LIN {X 0,Y 419.187,Z 570.974,A -85,B 0,C 180,E1 -10319.804,E2 -10319.804} C_VEL
LIN {X 0,Y 418.475,Z 578.407,A -85,B 0,C 180,E1 -10321.405,E2 -10321.405} C_VEL
LIN {X 0,Y 417.933,Z 584.546,A -85,B 0,C 180,E1 -10323.03,E2 -10323.03} C_VEL
LIN {X 0,Y 417.578,Z 589.288,A -85,B 0,C 180,E1 -10324.586,E2 -10324.586} C_VEL
LIN {X 0,Y 417.334,Z 593.011,A -85,B 0,C 180,E1 -10326.162,E2 -10326.162} C_VEL
LIN {X 0,Y 417.085,Z 596.065,A -85,B 0,C 180,E1 -10327.935,E2 -10327.935} C_VEL
LIN {X 0,Y 416.98,Z 597.612,A -85,B 0,C 180,E1 -10329.272,E2 -10329.272} C_VEL
LIN {X 0,Y 416.926,Z 598.729,A -85,B 0,C 180,E1 -10331.321,E2 -10331.321} C_VEL
LIN {X 0,Y 416.921,Z 598.396,A -85,B 0,C 180,E1 -10333.348,E2 -10333.348} C_VEL
LIN {X 0,Y 416.982,Z 596.643,A -85,B 0,C 180,E1 -10335.357,E2 -10335.357} C_VEL
LIN {X 0,Y 417.194,Z 593.458,A -85,B 0,C 180,E1 -10337.351,E2 -10337.351} C_VEL
LIN {X 0,Y 417.313,Z 591.479,A -85,B 0,C 180,E1 -10338.264,E2 -10338.264} C_VEL
LIN {X 0,Y 416.787,Z 589.683,A -85,B 0,C 180,E1 -10339.033,E2 -10339.033} C_VEL
LIN {X 0,Y 414.202,Z 586.34,A -85,B 0,C 180,E1 -10340.269,E2 -10340.269} C_VEL
LIN {X 0,Y 411.626,Z 582.374,A -85,B 0,C 180,E1 -10341.484,E2 -10341.484} C_VEL
LIN {X 0,Y 411.128,Z 579.597,A -85,B 0,C 180,E1 -10342.211,E2 -10342.211} C_VEL
LIN {X 0,Y 411.667,Z 572.14,A -85,B 0,C 180,E1 -10343.876,E2 -10343.876} C_VEL
LIN {X 0,Y 412.417,Z 564.039,A -85,B 0,C 180,E1 -10345.358,E2 -10345.358} C_VEL
LIN {X 0,Y 413.292,Z 554.296,A -85,B 0,C 180,E1 -10346.833,E2 -10346.833} C_VEL
LIN {X 0,Y 414.16,Z 543.524,A -85,B 0,C 180,E1 -10348.178,E2 -10348.178} C_VEL
LIN {X 0,Y 415.25,Z 531.337,A -85,B 0,C 180,E1 -10349.414,E2 -10349.414} C_VEL
LIN {X 0,Y 416.092,Z 519.779,A -85,B 0,C 180,E1 -10350.364,E2 -10350.364} C_VEL
LIN {X 0,Y 416.915,Z 506.934,A -85,B 0,C 180,E1 -10351.208,E2 -10351.208} C_VEL
LIN {X 0,Y 417.627,Z 493.022,A -85,B 0,C 180,E1 -10351.899,E2 -10351.899} C_VEL
LIN {X 0,Y 418.129,Z 479.426,A -85,B 0,C 180,E1 -10352.379,E2 -10352.379} C_VEL
LIN {X 0,Y 418.499,Z 462.629,A -85,B 0,C 180,E1 -10352.738,E2 -10352.738} C_VEL
LIN {X 0,Y 419.9,Z 361.135,A -85,B 0,C 180,E1 -10354.504,E2 -10354.504} C_VEL
LIN {X 0,Y 416.679,Z 347.393,A -85,B 0,C 180,E1 -10354.918,E2 -10354.918} C_VEL
LIN {X 0,Y 413.389,Z 338.049,A -85,B 0,C 180,E1 -10355.274,E2 -10355.274} C_VEL
LIN {X 0,Y 411.415,Z 327.865,A -85,B 0,C 180,E1 -10357.64,E2 -10357.64} C_VEL
LIN {X 0,Y 411.281,Z 327.882,A -85,B 0,C 180,E1 -10360.835,E2 -10360.835} C_VEL
LIN {X 0,Y 411.251,Z 327.88,A -85,B 0,C 180,E1 -10363.843,E2 -10363.843} C_VEL
LIN {X 0,Y 411.256,Z 327.881,A -85,B 0,C 180,E1 -10366.89,E2 -10366.89} C_VEL
LIN {X 0,Y 411.23,Z 327.882,A -85,B 0,C 180,E1 -10369.988,E2 -10369.988} C_VEL
LIN {X 0,Y 411.186,Z 327.894,A -85,B 0,C 180,E1 -10373.149,E2 -10373.149} C_VEL
LIN {X 0,Y 411.17,Z 327.89,A -85,B 0,C 180,E1 -10376.386,E2 -10376.386} C_VEL
LIN {X 0,Y 411.193,Z 327.887,A -85,B 0,C 180,E1 -10379.714,E2 -10379.714} C_VEL
LIN {X 0,Y 411.201,Z 327.89,A -85,B 0,C 180,E1 -10383.157,E2 -10383.157} C_VEL
LIN {X 0,Y 411.187,Z 327.89,A -85,B 0,C 180,E1 -10386.552,E2 -10386.552} C_VEL
LIN {X 0,Y 411.167,Z 327.889,A -85,B 0,C 180,E1 -10389.721,E2 -10389.721} C_VEL
LIN {X 0,Y 411.16,Z 327.893,A -85,B 0,C 180,E1 -10393.136,E2 -10393.136} C_VEL
LIN {X 0,Y 411.162,Z 327.89,A -85,B 0,C 180,E1 -10395.883,E2 -10395.883} C_VEL
LIN {X 0,Y 411.156,Z 327.891,A -85,B 0,C 180,E1 -10399.493,E2 -10399.493} C_VEL
LIN {X 0,Y 411.177,Z 327.889,A -85,B 0,C 180,E1 -10402.025,E2 -10402.025} C_VEL
LIN {X 0,Y 411.201,Z 327.886,A -85,B 0,C 180,E1 -10405.124,E2 -10405.124} C_VEL
LIN {X 0,Y 411.164,Z 327.891,A -85,B 0,C 180,E1 -10408.003,E2 -10408.003} C_VEL
LIN {X 0,Y 411.172,Z 327.889,A -85,B 0,C 180,E1 -10411.407,E2 -10411.407} C_VEL
LIN {X 0,Y 411.189,Z 327.888,A -85,B 0,C 180,E1 -10414.942,E2 -10414.942} C_VEL
LIN {X 0,Y 411.202,Z 327.887,A -85,B 0,C 180,E1 -10417.914,E2 -10417.914} C_VEL
LIN {X 0,Y 411.216,Z 327.884,A -85,B 0,C 180,E1 -10421.052,E2 -10421.052} C_VEL
LIN {X 0,Y 411.213,Z 327.889,A -85,B 0,C 180,E1 -10424.13,E2 -10424.13} C_VEL
LIN {X 0,Y 411.306,Z 327.872,A -85,B 0,C 180,E1 -10427.166,E2 -10427.166} C_VEL
LIN {X 0,Y 411.293,Z 327.881,A -85,B 0,C 180,E1 -10430.162,E2 -10430.162} C_VEL
LIN {X 0,Y 411.397,Z 327.861,A -85,B 0,C 180,E1 -10433.132,E2 -10433.132} C_VEL
LIN {X 0,Y 411.303,Z 327.872,A -85,B 0,C 180,E1 -10435.099,E2 -10435.099} C_VEL
LIN {X 0,Y 411.512,Z 327.853,A -85,B 0,C 180,E1 -10438.043,E2 -10438.043} C_VEL
LIN {X 0,Y 411.636,Z 327.838,A -85,B 0,C 180,E1 -10440,E2 -10440} C_VEL
LIN {X 0,Y 411.448,Z 327.854,A -85,B 0,C 180,E1 -10442.938,E2 -10442.938} C_VEL
LIN {X 0,Y 411.462,Z 327.86,A -85,B 0,C 180,E1 -10445.883,E2 -10445.883} C_VEL
LIN {X 0,Y 411.337,Z 327.868,A -85,B 0,C 180,E1 -10448.846,E2 -10448.846} C_VEL
LIN {X 0,Y 411.287,Z 327.881,A -85,B 0,C 180,E1 -10451.833,E2 -10451.833} C_VEL
LIN {X 0,Y 411.263,Z 327.877,A -85,B 0,C 180,E1 -10454.853,E2 -10454.853} C_VEL
LIN {X 0,Y 411.256,Z 327.883,A -85,B 0,C 180,E1 -10457.915,E2 -10457.915} C_VEL
LIN {X 0,Y 411.201,Z 327.886,A -85,B 0,C 180,E1 -10461.034,E2 -10461.034} C_VEL
LIN {X 0,Y 411.23,Z 327.882,A -85,B 0,C 180,E1 -10464.216,E2 -10464.216} C_VEL
LIN {X 0,Y 411.263,Z 327.884,A -85,B 0,C 180,E1 -10467.478,E2 -10467.478} C_VEL
LIN {X 0,Y 411.193,Z 327.887,A -85,B 0,C 180,E1 -10470.848,E2 -10470.848} C_VEL
LIN {X 0,Y 411.209,Z 327.884,A -85,B 0,C 180,E1 -10474.333,E2 -10474.333} C_VEL
LIN {X 0,Y 411.199,Z 327.886,A -85,B 0,C 180,E1 -10477.974,E2 -10477.974} C_VEL
LIN {X 0,Y 411.186,Z 327.887,A -85,B 0,C 180,E1 -10480.504,E2 -10480.504} C_VEL
LIN {X 0,Y 411.181,Z 327.893,A -85,B 0,C 180,E1 -10483.133,E2 -10483.133} C_VEL
LIN {X 0,Y 411.173,Z 327.889,A -85,B 0,C 180,E1 -10485.881,E2 -10485.881} C_VEL
LIN {X 0,Y 411.167,Z 327.892,A -85,B 0,C 180,E1 -10488.771,E2 -10488.771} C_VEL
LIN {X 0,Y 411.209,Z 327.885,A -85,B 0,C 180,E1 -10491.831,E2 -10491.831} C_VEL
LIN {X 0,Y 411.215,Z 327.89,A -85,B 0,C 180,E1 -10495.121,E2 -10495.121} C_VEL
LIN {X 0,Y 411.17,Z 327.895,A -85,B 0,C 180,E1 -10498.002,E2 -10498.002} C_VEL
LIN {X 0,Y 411.253,Z 327.986,A -85,B 0,C 180,E1 -10499.548,E2 -10499.548} C_VEL
LIN {X 0,Y 415.143,Z 345.403,A -85,B 0,C 180,E1 -10503.042,E2 -10503.042} C_VEL
LIN {X 0,Y 415.639,Z 350.042,A -85,B 0,C 180,E1 -10503.919,E2 -10503.919} C_VEL
LIN {X 0,Y 414.463,Z 366.202,A -85,B 0,C 180,E1 -10506.786,E2 -10506.786} C_VEL
LIN {X 0,Y 419.646,Z 398,A -85,B 0,C 180,E1 -10507.644,E2 -10507.644} C_VEL
LIN {X 0,Y 417.994,Z 504.817,A -85,B 0,C 180,E1 -10509.516,E2 -10509.516} C_VEL
LIN {X 0,Y 417.425,Z 519.405,A -85,B 0,C 180,E1 -10509.969,E2 -10509.969} C_VEL
LIN {X 0,Y 416.661,Z 532.568,A -85,B 0,C 180,E1 -10510.558,E2 -10510.558} C_VEL
LIN {X 0,Y 415.788,Z 546.414,A -85,B 0,C 180,E1 -10511.394,E2 -10511.394} C_VEL
LIN {X 0,Y 414.754,Z 559.052,A -85,B 0,C 180,E1 -10512.368,E2 -10512.368} C_VEL
LIN {X 0,Y 413.786,Z 570.591,A -85,B 0,C 180,E1 -10513.471,E2 -10513.471} C_VEL
LIN {X 0,Y 412.832,Z 581.181,A -85,B 0,C 180,E1 -10514.699,E2 -10514.699} C_VEL
LIN {X 0,Y 412.026,Z 591.716,A -85,B 0,C 180,E1 -10516.183,E2 -10516.183} C_VEL
LIN {X 0,Y 411.345,Z 600.394,A -85,B 0,C 180,E1 -10517.668,E2 -10517.668} C_VEL
LIN {X 0,Y 410.689,Z 608.675,A -85,B 0,C 180,E1 -10519.399,E2 -10519.399} C_VEL
LIN {X 0,Y 410.326,Z 615.336,A -85,B 0,C 180,E1 -10521.132,E2 -10521.132} C_VEL
LIN {X 0,Y 410.062,Z 621.237,A -85,B 0,C 180,E1 -10523.109,E2 -10523.109} C_VEL
LIN {X 0,Y 409.983,Z 625.54,A -85,B 0,C 180,E1 -10525.082,E2 -10525.082} C_VEL
LIN {X 0,Y 409.955,Z 628.378,A -85,B 0,C 180,E1 -10527.051,E2 -10527.051} C_VEL
LIN {X 0,Y 409.954,Z 629.831,A -85,B 0,C 180,E1 -10529.017,E2 -10529.017} C_VEL
LIN {X 0,Y 409.954,Z 629.934,A -85,B 0,C 180,E1 -10530.981,E2 -10530.981} C_VEL
LIN {X 0,Y 409.994,Z 629.483,A -85,B 0,C 180,E1 -10531.964,E2 -10531.964} C_VEL
LIN {X 0,Y 409.922,Z 627.565,A -85,B 0,C 180,E1 -10533.931,E2 -10533.931} C_VEL
LIN {X 0,Y 410.015,Z 624.244,A -85,B 0,C 180,E1 -10535.902,E2 -10535.902} C_VEL
LIN {X 0,Y 410.154,Z 620.769,A -85,B 0,C 180,E1 -10537.383,E2 -10537.383} C_VEL
LIN {X 0,Y 410.472,Z 614.788,A -85,B 0,C 180,E1 -10539.36,E2 -10539.36} C_VEL
LIN {X 0,Y 410.951,Z 608.074,A -85,B 0,C 180,E1 -10541.092,E2 -10541.092} C_VEL
LIN {X 0,Y 411.639,Z 599.741,A -85,B 0,C 180,E1 -10542.823,E2 -10542.823} C_VEL
LIN {X 0,Y 412.437,Z 591.079,A -85,B 0,C 180,E1 -10544.304,E2 -10544.304} C_VEL
LIN {X 0,Y 413.43,Z 580.609,A -85,B 0,C 180,E1 -10545.782,E2 -10545.782} C_VEL
LIN {X 0,Y 414.659,Z 568.924,A -85,B 0,C 180,E1 -10547.126,E2 -10547.126} C_VEL
LIN {X 0,Y 415.755,Z 557.26,A -85,B 0,C 180,E1 -10548.223,E2 -10548.223} C_VEL
LIN {X 0,Y 416.929,Z 544.33,A -85,B 0,C 180,E1 -10549.197,E2 -10549.197} C_VEL
LIN {X 0,Y 417.819,Z 531.185,A -85,B 0,C 180,E1 -10549.978,E2 -10549.978} C_VEL
LIN {X 0,Y 418.734,Z 517.564,A -85,B 0,C 180,E1 -10550.573,E2 -10550.573} C_VEL
LIN {X 0,Y 419.385,Z 503.626,A -85,B 0,C 180,E1 -10550.989,E2 -10550.989} C_VEL
LIN {X 0,Y 421.169,Z 397.55,A -85,B 0,C 180,E1 -10552.879,E2 -10552.879} C_VEL
LIN {X 0,Y 416.853,Z 373.266,A -85,B 0,C 180,E1 -10553.621,E2 -10553.621} C_VEL
LIN {X 0,Y 415.311,Z 365.541,A -85,B 0,C 180,E1 -10553.906,E2 -10553.906} C_VEL
LIN {X 0,Y 416.42,Z 351.139,A -85,B 0,C 180,E1 -10556.556,E2 -10556.556} C_VEL
LIN {X 0,Y 414.822,Z 342.635,A -85,B 0,C 180,E1 -10558.318,E2 -10558.318} C_VEL
LIN {X 0,Y 412.132,Z 331.458,A -85,B 0,C 180,E1 -10560.768,E2 -10560.768} C_VEL
LIN {X 0,Y 411.159,Z 327.894,A -85,B 0,C 180,E1 -10561.594,E2 -10561.594} C_VEL
LIN {X 0,Y 411.209,Z 327.892,A -85,B 0,C 180,E1 -10564.878,E2 -10564.878} C_VEL
LIN {X 0,Y 411.211,Z 327.886,A -85,B 0,C 180,E1 -10568.169,E2 -10568.169} C_VEL
LIN {X 0,Y 411.196,Z 327.885,A -85,B 0,C 180,E1 -10571.233,E2 -10571.233} C_VEL
LIN {X 0,Y 411.173,Z 327.893,A -85,B 0,C 180,E1 -10574.489,E2 -10574.489} C_VEL
LIN {X 0,Y 411.179,Z 327.893,A -85,B 0,C 180,E1 -10578.194,E2 -10578.194} C_VEL
LIN {X 0,Y 411.213,Z 327.876,A -85,B 0,C 180,E1 -10580.775,E2 -10580.775} C_VEL
LIN {X 0,Y 411.194,Z 327.889,A -85,B 0,C 180,E1 -10584.47,E2 -10584.47} C_VEL
LIN {X 0,Y 411.162,Z 327.891,A -85,B 0,C 180,E1 -10588.002,E2 -10588.002} C_VEL
LIN {X 0,Y 411.217,Z 327.884,A -85,B 0,C 180,E1 -10591.41,E2 -10591.41} C_VEL
LIN {X 0,Y 411.229,Z 327.885,A -85,B 0,C 180,E1 -10594.706,E2 -10594.706} C_VEL
LIN {X 0,Y 411.197,Z 327.885,A -85,B 0,C 180,E1 -10597.913,E2 -10597.913} C_VEL
LIN {X 0,Y 411.217,Z 327.878,A -85,B 0,C 180,E1 -10601.051,E2 -10601.051} C_VEL
LIN {X 0,Y 411.255,Z 327.879,A -85,B 0,C 180,E1 -10604.131,E2 -10604.131} C_VEL
LIN {X 0,Y 411.295,Z 327.875,A -85,B 0,C 180,E1 -10607.165,E2 -10607.165} C_VEL
LIN {X 0,Y 411.282,Z 327.88,A -85,B 0,C 180,E1 -10610.161,E2 -10610.161} C_VEL
LIN {X 0,Y 411.474,Z 327.851,A -85,B 0,C 180,E1 -10612.146,E2 -10612.146} C_VEL
LIN {X 0,Y 411.462,Z 327.857,A -85,B 0,C 180,E1 -10614.117,E2 -10614.117} C_VEL
LIN {X 0,Y 411.494,Z 327.852,A -85,B 0,C 180,E1 -10618.042,E2 -10618.042} C_VEL
LIN {X 0,Y 411.368,Z 327.863,A -85,B 0,C 180,E1 -10620.979,E2 -10620.979} C_VEL
LIN {X 0,Y 411.435,Z 327.857,A -85,B 0,C 180,E1 -10622.937,E2 -10622.937} C_VEL
LIN {X 0,Y 411.375,Z 327.865,A -85,B 0,C 180,E1 -10626.868,E2 -10626.868} C_VEL
LIN {X 0,Y 411.27,Z 327.88,A -85,B 0,C 180,E1 -10629.839,E2 -10629.839} C_VEL
LIN {X 0,Y 411.296,Z 327.873,A -85,B 0,C 180,E1 -10633.104,E2 -10633.104} C_VEL
LIN {X 0,Y 411.247,Z 327.879,A -85,B 0,C 180,E1 -10636.889,E2 -10636.889} C_VEL
LIN {X 0,Y 411.221,Z 327.885,A -85,B 0,C 180,E1 -10639.987,E2 -10639.987} C_VEL
LIN {X 0,Y 411.191,Z 327.89,A -85,B 0,C 180,E1 -10643.148,E2 -10643.148} C_VEL
LIN {X 0,Y 411.176,Z 327.892,A -85,B 0,C 180,E1 -10646.385,E2 -10646.385} C_VEL
LIN {X 0,Y 411.187,Z 327.889,A -85,B 0,C 180,E1 -10649.713,E2 -10649.713} C_VEL
LIN {X 0,Y 411.197,Z 327.885,A -85,B 0,C 180,E1 -10653.156,E2 -10653.156} C_VEL
LIN {X 0,Y 411.183,Z 327.888,A -85,B 0,C 180,E1 -10656.553,E2 -10656.553} C_VEL
LIN {X 0,Y 411.2,Z 327.884,A -85,B 0,C 180,E1 -10659.728,E2 -10659.728} C_VEL
LIN {X 0,Y 411.164,Z 327.896,A -85,B 0,C 180,E1 -10663.134,E2 -10663.134} C_VEL
LIN {X 0,Y 411.202,Z 327.999,A -85,B 0,C 180,E1 -10665.36,E2 -10665.36} C_VEL
LIN {X 0,Y 413.682,Z 338.677,A -85,B 0,C 180,E1 -10668.055,E2 -10668.055} C_VEL
LIN {X 0,Y 419.545,Z 352.95,A -85,B 0,C 180,E1 -10668.744,E2 -10668.744} C_VEL
LIN {X 0,Y 421.668,Z 362.235,A -85,B 0,C 180,E1 -10669.061,E2 -10669.061} C_VEL
LIN {X 0,Y 419.69,Z 475.315,A -85,B 0,C 180,E1 -10671.082,E2 -10671.082} C_VEL
LIN {X 0,Y 419.118,Z 489.735,A -85,B 0,C 180,E1 -10671.539,E2 -10671.539} C_VEL
LIN {X 0,Y 418.491,Z 502.416,A -85,B 0,C 180,E1 -10672.12,E2 -10672.12} C_VEL
LIN {X 0,Y 417.635,Z 514.875,A -85,B 0,C 180,E1 -10672.866,E2 -10672.866} C_VEL
LIN {X 0,Y 416.65,Z 527.347,A -85,B 0,C 180,E1 -10673.818,E2 -10673.818} C_VEL
LIN {X 0,Y 415.532,Z 538.826,A -85,B 0,C 180,E1 -10674.898,E2 -10674.898} C_VEL
LIN {X 0,Y 414.456,Z 550.011,A -85,B 0,C 180,E1 -10676.191,E2 -10676.191} C_VEL
LIN {X 0,Y 413.412,Z 560.201,A -85,B 0,C 180,E1 -10677.624,E2 -10677.624} C_VEL
LIN {X 0,Y 412.46,Z 569.724,A -85,B 0,C 180,E1 -10679.259,E2 -10679.259} C_VEL
LIN {X 0,Y 411.627,Z 577.758,A -85,B 0,C 180,E1 -10680.957,E2 -10680.957} C_VEL
LIN {X 0,Y 410.958,Z 584.641,A -85,B 0,C 180,E1 -10682.782,E2 -10682.782} C_VEL
LIN {X 0,Y 410.506,Z 590.156,A -85,B 0,C 180,E1 -10684.66,E2 -10684.66} C_VEL
LIN {X 0,Y 410.229,Z 593.767,A -85,B 0,C 180,E1 -10686.26,E2 -10686.26} C_VEL
LIN {X 0,Y 410.012,Z 596.36,A -85,B 0,C 180,E1 -10687.847,E2 -10687.847} C_VEL
LIN {X 0,Y 409.867,Z 598.478,A -85,B 0,C 180,E1 -10689.945,E2 -10689.945} C_VEL
LIN {X 0,Y 409.851,Z 598.955,A -85,B 0,C 180,E1 -10690.987,E2 -10690.987} C_VEL
LIN {X 0,Y 409.812,Z 598.808,A -85,B 0,C 180,E1 -10693.051,E2 -10693.051} C_VEL
LIN {X 0,Y 409.898,Z 597.235,A -85,B 0,C 180,E1 -10695.098,E2 -10695.098} C_VEL
LIN {X 0,Y 410.087,Z 594.236,A -85,B 0,C 180,E1 -10697.128,E2 -10697.128} C_VEL
LIN {X 0,Y 410.394,Z 589.754,A -85,B 0,C 180,E1 -10699.143,E2 -10699.143} C_VEL
LIN {X 0,Y 410.654,Z 585.313,A -85,B 0,C 180,E1 -10700.644,E2 -10700.644} C_VEL
LIN {X 0,Y 411.128,Z 579.597,A -85,B 0,C 180,E1 -10702.211,E2 -10702.211} C_VEL
LIN {X 0,Y 410.657,Z 576.696,A -85,B 0,C 180,E1 -10702.924,E2 -10702.924} C_VEL
LIN {X 0,Y 408.241,Z 571.685,A -85,B 0,C 180,E1 -10704.076,E2 -10704.076} C_VEL
LIN {X 0,Y 405.915,Z 566.26,A -85,B 0,C 180,E1 -10705.195,E2 -10705.195} C_VEL
LIN {X 0,Y 405.587,Z 562.534,A -85,B 0,C 180,E1 -10705.847,E2 -10705.847} C_VEL
LIN {X 0,Y 406.525,Z 552.936,A -85,B 0,C 180,E1 -10707.276,E2 -10707.276} C_VEL
LIN {X 0,Y 407.406,Z 542.887,A -85,B 0,C 180,E1 -10708.519,E2 -10708.519} C_VEL
LIN {X 0,Y 408.408,Z 531.578,A -85,B 0,C 180,E1 -10709.674,E2 -10709.674} C_VEL
LIN {X 0,Y 409.363,Z 518.69,A -85,B 0,C 180,E1 -10710.739,E2 -10710.739} C_VEL
LIN {X 0,Y 410.306,Z 505.333,A -85,B 0,C 180,E1 -10711.596,E2 -10711.596} C_VEL
LIN {X 0,Y 410.914,Z 492.304,A -85,B 0,C 180,E1 -10712.237,E2 -10712.237} C_VEL
LIN {X 0,Y 411.405,Z 479.337,A -85,B 0,C 180,E1 -10712.693,E2 -10712.693} C_VEL
LIN {X 0,Y 411.795,Z 462.325,A -85,B 0,C 180,E1 -10713.058,E2 -10713.058} C_VEL
LIN {X 0,Y 413.256,Z 362.392,A -85,B 0,C 180,E1 -10714.82,E2 -10714.82} C_VEL
LIN {X 0,Y 410.291,Z 349.7,A -85,B 0,C 180,E1 -10715.211,E2 -10715.211} C_VEL
LIN {X 0,Y 406.245,Z 338.279,A -85,B 0,C 180,E1 -10715.663,E2 -10715.663} C_VEL
LIN {X 0,Y 404.372,Z 328.745,A -85,B 0,C 180,E1 -10717.944,E2 -10717.944} C_VEL
LIN {X 0,Y 404.248,Z 328.758,A -85,B 0,C 180,E1 -10721.026,E2 -10721.026} C_VEL
LIN {X 0,Y 404.207,Z 328.756,A -85,B 0,C 180,E1 -10724.089,E2 -10724.089} C_VEL
LIN {X 0,Y 404.201,Z 328.764,A -85,B 0,C 180,E1 -10727.193,E2 -10727.193} C_VEL
LIN {X 0,Y 404.163,Z 328.762,A -85,B 0,C 180,E1 -10730.352,E2 -10730.352} C_VEL
LIN {X 0,Y 404.147,Z 328.766,A -85,B 0,C 180,E1 -10733.577,E2 -10733.577} C_VEL
LIN {X 0,Y 404.102,Z 328.774,A -85,B 0,C 180,E1 -10736.885,E2 -10736.885} C_VEL
LIN {X 0,Y 404.139,Z 328.765,A -85,B 0,C 180,E1 -10740.286,E2 -10740.286} C_VEL
LIN {X 0,Y 404.135,Z 328.765,A -85,B 0,C 180,E1 -10743.814,E2 -10743.814} C_VEL
LIN {X 0,Y 404.13,Z 328.773,A -85,B 0,C 180,E1 -10746.874,E2 -10746.874} C_VEL
LIN {X 0,Y 404.116,Z 328.768,A -85,B 0,C 180,E1 -10750.075,E2 -10750.075} C_VEL
LIN {X 0,Y 404.14,Z 328.768,A -85,B 0,C 180,E1 -10753.082,E2 -10753.082} C_VEL
LIN {X 0,Y 404.119,Z 328.767,A -85,B 0,C 180,E1 -10755.923,E2 -10755.923} C_VEL
LIN {X 0,Y 404.101,Z 328.776,A -85,B 0,C 180,E1 -10758.633,E2 -10758.633} C_VEL
LIN {X 0,Y 404.133,Z 328.766,A -85,B 0,C 180,E1 -10761.497,E2 -10761.497} C_VEL
LIN {X 0,Y 404.176,Z 328.763,A -85,B 0,C 180,E1 -10764.984,E2 -10764.984} C_VEL
LIN {X 0,Y 404.139,Z 328.771,A -85,B 0,C 180,E1 -10768.443,E2 -10768.443} C_VEL
LIN {X 0,Y 404.15,Z 328.766,A -85,B 0,C 180,E1 -10770.863,E2 -10770.863} C_VEL
LIN {X 0,Y 404.154,Z 328.766,A -85,B 0,C 180,E1 -10774.723,E2 -10774.723} C_VEL
LIN {X 0,Y 404.166,Z 328.761,A -85,B 0,C 180,E1 -10777.508,E2 -10777.508} C_VEL
LIN {X 0,Y 404.161,Z 328.765,A -85,B 0,C 180,E1 -10780.708,E2 -10780.708} C_VEL
LIN {X 0,Y 404.183,Z 328.762,A -85,B 0,C 180,E1 -10783.847,E2 -10783.847} C_VEL
LIN {X 0,Y 404.286,Z 328.747,A -85,B 0,C 180,E1 -10786.939,E2 -10786.939} C_VEL
LIN {X 0,Y 404.258,Z 328.755,A -85,B 0,C 180,E1 -10789.989,E2 -10789.989} C_VEL
LIN {X 0,Y 404.346,Z 328.739,A -85,B 0,C 180,E1 -10793.012,E2 -10793.012} C_VEL
LIN {X 0,Y 404.274,Z 328.748,A -85,B 0,C 180,E1 -10795.014,E2 -10795.014} C_VEL
LIN {X 0,Y 404.481,Z 328.729,A -85,B 0,C 180,E1 -10798.009,E2 -10798.009} C_VEL
LIN {X 0,Y 404.606,Z 328.714,A -85,B 0,C 180,E1 -10800,E2 -10800} C_VEL
LIN {X 0,Y 404.406,Z 328.731,A -85,B 0,C 180,E1 -10802.989,E2 -10802.989} C_VEL
LIN {X 0,Y 404.409,Z 328.737,A -85,B 0,C 180,E1 -10805.985,E2 -10805.985} C_VEL
LIN {X 0,Y 404.279,Z 328.747,A -85,B 0,C 180,E1 -10809.002,E2 -10809.002} C_VEL
LIN {X 0,Y 404.259,Z 328.754,A -85,B 0,C 180,E1 -10812.042,E2 -10812.042} C_VEL
LIN {X 0,Y 404.21,Z 328.757,A -85,B 0,C 180,E1 -10815.118,E2 -10815.118} C_VEL
LIN {X 0,Y 404.214,Z 328.757,A -85,B 0,C 180,E1 -10818.238,E2 -10818.238} C_VEL
LIN {X 0,Y 404.164,Z 328.766,A -85,B 0,C 180,E1 -10821.418,E2 -10821.418} C_VEL
LIN {X 0,Y 404.181,Z 328.76,A -85,B 0,C 180,E1 -10824.666,E2 -10824.666} C_VEL
LIN {X 0,Y 404.199,Z 328.759,A -85,B 0,C 180,E1 -10828,E2 -10828} C_VEL
LIN {X 0,Y 404.144,Z 328.77,A -85,B 0,C 180,E1 -10831.558,E2 -10831.558} C_VEL
LIN {X 0,Y 404.188,Z 328.761,A -85,B 0,C 180,E1 -10835.016,E2 -10835.016} C_VEL
LIN {X 0,Y 404.159,Z 328.763,A -85,B 0,C 180,E1 -10838.757,E2 -10838.757} C_VEL
LIN {X 0,Y 404.128,Z 328.77,A -85,B 0,C 180,E1 -10841.6,E2 -10841.6} C_VEL
LIN {X 0,Y 404.153,Z 328.764,A -85,B 0,C 180,E1 -10844.522,E2 -10844.522} C_VEL
LIN {X 0,Y 404.14,Z 328.771,A -85,B 0,C 180,E1 -10847.295,E2 -10847.295} C_VEL
LIN {X 0,Y 404.173,Z 328.761,A -85,B 0,C 180,E1 -10849.955,E2 -10849.955} C_VEL
LIN {X 0,Y 404.141,Z 328.772,A -85,B 0,C 180,E1 -10853.125,E2 -10853.125} C_VEL
LIN {X 0,Y 404.149,Z 328.764,A -85,B 0,C 180,E1 -10856.187,E2 -10856.187} C_VEL
LIN {X 0,Y 404.206,Z 328.866,A -85,B 0,C 180,E1 -10859.249,E2 -10859.249} C_VEL
LIN {X 0,Y 407.814,Z 344.98,A -85,B 0,C 180,E1 -10862.548,E2 -10862.548} C_VEL
LIN {X 0,Y 408.745,Z 350.969,A -85,B 0,C 180,E1 -10863.72,E2 -10863.72} C_VEL
LIN {X 0,Y 407.605,Z 366.006,A -85,B 0,C 180,E1 -10866.432,E2 -10866.432} C_VEL
LIN {X 0,Y 412.925,Z 398.004,A -85,B 0,C 180,E1 -10867.309,E2 -10867.309} C_VEL
LIN {X 0,Y 411.279,Z 504.184,A -85,B 0,C 180,E1 -10869.199,E2 -10869.199} C_VEL
LIN {X 0,Y 410.714,Z 518.13,A -85,B 0,C 180,E1 -10869.627,E2 -10869.627} C_VEL
LIN {X 0,Y 409.928,Z 531.687,A -85,B 0,C 180,E1 -10870.234,E2 -10870.234} C_VEL
LIN {X 0,Y 409.063,Z 544.802,A -85,B 0,C 180,E1 -10871.021,E2 -10871.021} C_VEL
LIN {X 0,Y 407.941,Z 558.312,A -85,B 0,C 180,E1 -10872.063,E2 -10872.063} C_VEL
LIN {X 0,Y 406.902,Z 569.932,A -85,B 0,C 180,E1 -10873.183,E2 -10873.183} C_VEL
LIN {X 0,Y 405.925,Z 580.59,A -85,B 0,C 180,E1 -10874.433,E2 -10874.433} C_VEL
LIN {X 0,Y 405.054,Z 591.177,A -85,B 0,C 180,E1 -10875.941,E2 -10875.941} C_VEL
LIN {X 0,Y 404.375,Z 599.905,A -85,B 0,C 180,E1 -10877.452,E2 -10877.452} C_VEL
LIN {X 0,Y 403.665,Z 608.245,A -85,B 0,C 180,E1 -10879.212,E2 -10879.212} C_VEL
LIN {X 0,Y 403.274,Z 614.944,A -85,B 0,C 180,E1 -10880.975,E2 -10880.975} C_VEL
LIN {X 0,Y 402.985,Z 620.877,A -85,B 0,C 180,E1 -10882.987,E2 -10882.987} C_VEL
LIN {X 0,Y 402.895,Z 625.208,A -85,B 0,C 180,E1 -10884.996,E2 -10884.996} C_VEL
LIN {X 0,Y 402.854,Z 628.07,A -85,B 0,C 180,E1 -10886.999,E2 -10886.999} C_VEL
LIN {X 0,Y 402.928,Z 628.981,A -85,B 0,C 180,E1 -10888,E2 -10888} C_VEL
LIN {X 0,Y 402.87,Z 629.776,A -85,B 0,C 180,E1 -10889.999,E2 -10889.999} C_VEL
LIN {X 0,Y 402.905,Z 629.23,A -85,B 0,C 180,E1 -10891.998,E2 -10891.998} C_VEL
LIN {X 0,Y 402.841,Z 627.337,A -85,B 0,C 180,E1 -10894.001,E2 -10894.001} C_VEL
LIN {X 0,Y 402.938,Z 624.051,A -85,B 0,C 180,E1 -10896.006,E2 -10896.006} C_VEL
LIN {X 0,Y 403.06,Z 620.591,A -85,B 0,C 180,E1 -10897.513,E2 -10897.513} C_VEL
LIN {X 0,Y 403.422,Z 614.638,A -85,B 0,C 180,E1 -10899.525,E2 -10899.525} C_VEL
LIN {X 0,Y 403.96,Z 607.958,A -85,B 0,C 180,E1 -10901.286,E2 -10901.286} C_VEL
LIN {X 0,Y 404.687,Z 599.672,A -85,B 0,C 180,E1 -10903.047,E2 -10903.047} C_VEL
LIN {X 0,Y 405.524,Z 591.051,A -85,B 0,C 180,E1 -10904.553,E2 -10904.553} C_VEL
LIN {X 0,Y 406.581,Z 580.64,A -85,B 0,C 180,E1 -10906.054,E2 -10906.054} C_VEL
LIN {X 0,Y 407.884,Z 569.037,A -85,B 0,C 180,E1 -10907.419,E2 -10907.419} C_VEL
LIN {X 0,Y 409.026,Z 557.478,A -85,B 0,C 180,E1 -10908.533,E2 -10908.533} C_VEL
LIN {X 0,Y 410.188,Z 545.227,A -85,B 0,C 180,E1 -10909.486,E2 -10909.486} C_VEL
LIN {X 0,Y 411.193,Z 531.73,A -85,B 0,C 180,E1 -10910.314,E2 -10910.314} C_VEL
LIN {X 0,Y 412.174,Z 517.641,A -85,B 0,C 180,E1 -10910.948,E2 -10910.948} C_VEL
LIN {X 0,Y 412.867,Z 503.924,A -85,B 0,C 180,E1 -10911.369,E2 -10911.369} C_VEL
LIN {X 0,Y 414.684,Z 398.141,A -85,B 0,C 180,E1 -10913.291,E2 -10913.291} C_VEL
LIN {X 0,Y 410.617,Z 375.165,A -85,B 0,C 180,E1 -10914.012,E2 -10914.012} C_VEL
LIN {X 0,Y 408.563,Z 365.279,A -85,B 0,C 180,E1 -10914.382,E2 -10914.382} C_VEL
LIN {X 0,Y 409.619,Z 353.967,A -85,B 0,C 180,E1 -10916.492,E2 -10916.492} C_VEL
LIN {X 0,Y 409.34,Z 350.747,A -85,B 0,C 180,E1 -10917.14,E2 -10917.14} C_VEL
LIN {X 0,Y 406.522,Z 338.085,A -85,B 0,C 180,E1 -10919.895,E2 -10919.895} C_VEL
LIN {X 0,Y 404.117,Z 328.77,A -85,B 0,C 180,E1 -10922.045,E2 -10922.045} C_VEL
LIN {X 0,Y 404.179,Z 328.764,A -85,B 0,C 180,E1 -10925.189,E2 -10925.189} C_VEL
LIN {X 0,Y 404.16,Z 328.761,A -85,B 0,C 180,E1 -10928.755,E2 -10928.755} C_VEL
LIN {X 0,Y 404.146,Z 328.761,A -85,B 0,C 180,E1 -10931.603,E2 -10931.603} C_VEL
LIN {X 0,Y 404.142,Z 328.768,A -85,B 0,C 180,E1 -10934.521,E2 -10934.521} C_VEL
LIN {X 0,Y 404.135,Z 328.769,A -85,B 0,C 180,E1 -10937.295,E2 -10937.295} C_VEL
LIN {X 0,Y 404.163,Z 328.754,A -85,B 0,C 180,E1 -10939.954,E2 -10939.954} C_VEL
LIN {X 0,Y 404.134,Z 328.768,A -85,B 0,C 180,E1 -10943.123,E2 -10943.123} C_VEL
LIN {X 0,Y 404.139,Z 328.771,A -85,B 0,C 180,E1 -10946.187,E2 -10946.187} C_VEL
LIN {X 0,Y 404.148,Z 328.765,A -85,B 0,C 180,E1 -10949.715,E2 -10949.715} C_VEL
LIN {X 0,Y 404.188,Z 328.757,A -85,B 0,C 180,E1 -10953.122,E2 -10953.122} C_VEL
LIN {X 0,Y 404.167,Z 328.763,A -85,B 0,C 180,E1 -10955.333,E2 -10955.333} C_VEL
LIN {X 0,Y 404.152,Z 328.768,A -85,B 0,C 180,E1 -10958.581,E2 -10958.581} C_VEL
LIN {X 0,Y 404.203,Z 328.755,A -85,B 0,C 180,E1 -10961.761,E2 -10961.761} C_VEL
LIN {X 0,Y 404.203,Z 328.752,A -85,B 0,C 180,E1 -10964.882,E2 -10964.882} C_VEL
LIN {X 0,Y 404.247,Z 328.753,A -85,B 0,C 180,E1 -10967.958,E2 -10967.958} C_VEL
LIN {X 0,Y 404.425,Z 328.729,A -85,B 0,C 180,E1 -10972.099,E2 -10972.099} C_VEL
LIN {X 0,Y 404.411,Z 328.733,A -85,B 0,C 180,E1 -10974.015,E2 -10974.015} C_VEL
LIN {X 0,Y 404.463,Z 328.727,A -85,B 0,C 180,E1 -10978.008,E2 -10978.008} C_VEL
LIN {X 0,Y 404.338,Z 328.738,A -85,B 0,C 180,E1 -10980.996,E2 -10980.996} C_VEL
LIN {X 0,Y 404.394,Z 328.735,A -85,B 0,C 180,E1 -10982.988,E2 -10982.988} C_VEL
LIN {X 0,Y 404.326,Z 328.744,A -85,B 0,C 180,E1 -10986.988,E2 -10986.988} C_VEL
LIN {X 0,Y 404.238,Z 328.756,A -85,B 0,C 180,E1 -10990.012,E2 -10990.012} C_VEL
LIN {X 0,Y 404.257,Z 328.75,A -85,B 0,C 180,E1 -10993.211,E2 -10993.211} C_VEL
LIN {X 0,Y 404.206,Z 328.757,A -85,B 0,C 180,E1 -10997.007,E2 -10997.007} C_VEL
LIN {X 0,Y 404.154,Z 328.764,A -85,B 0,C 180,E1 -11000.352,E2 -11000.352} C_VEL
LIN {X 0,Y 404.152,Z 328.768,A -85,B 0,C 180,E1 -11003.575,E2 -11003.575} C_VEL
LIN {X 0,Y 404.119,Z 328.774,A -85,B 0,C 180,E1 -11006.882,E2 -11006.882} C_VEL
LIN {X 0,Y 404.134,Z 328.77,A -85,B 0,C 180,E1 -11010.286,E2 -11010.286} C_VEL
LIN {X 0,Y 404.135,Z 328.769,A -85,B 0,C 180,E1 -11013.813,E2 -11013.813} C_VEL
LIN {X 0,Y 404.126,Z 328.766,A -85,B 0,C 180,E1 -11016.875,E2 -11016.875} C_VEL
LIN {X 0,Y 404.139,Z 328.766,A -85,B 0,C 180,E1 -11020.081,E2 -11020.081} C_VEL
LIN {X 0,Y 404.144,Z 328.771,A -85,B 0,C 180,E1 -11023.084,E2 -11023.084} C_VEL
LIN {X 0,Y 404.173,Z 328.833,A -85,B 0,C 180,E1 -11024.915,E2 -11024.915} C_VEL
LIN {X 0,Y 406.563,Z 339.112,A -85,B 0,C 180,E1 -11027.551,E2 -11027.551} C_VEL
LIN {X 0,Y 413.427,Z 355.249,A -85,B 0,C 180,E1 -11028.368,E2 -11028.368} C_VEL
LIN {X 0,Y 415.281,Z 363.841,A -85,B 0,C 180,E1 -11028.663,E2 -11028.663} C_VEL
LIN {X 0,Y 413.206,Z 475.522,A -85,B 0,C 180,E1 -11030.688,E2 -11030.688} C_VEL
LIN {X 0,Y 412.609,Z 490.01,A -85,B 0,C 180,E1 -11031.153,E2 -11031.153} C_VEL
LIN {X 0,Y 411.918,Z 503.176,A -85,B 0,C 180,E1 -11031.769,E2 -11031.769} C_VEL
LIN {X 0,Y 410.923,Z 516.825,A -85,B 0,C 180,E1 -11032.617,E2 -11032.617} C_VEL
LIN {X 0,Y 409.835,Z 529.409,A -85,B 0,C 180,E1 -11033.621,E2 -11033.621} C_VEL
LIN {X 0,Y 408.618,Z 541.49,A -85,B 0,C 180,E1 -11034.819,E2 -11034.819} C_VEL
LIN {X 0,Y 407.535,Z 551.904,A -85,B 0,C 180,E1 -11036.086,E2 -11036.086} C_VEL
LIN {X 0,Y 406.409,Z 562.075,A -85,B 0,C 180,E1 -11037.584,E2 -11037.584} C_VEL
LIN {X 0,Y 405.399,Z 571.242,A -85,B 0,C 180,E1 -11039.243,E2 -11039.243} C_VEL
LIN {X 0,Y 404.586,Z 578.728,A -85,B 0,C 180,E1 -11040.898,E2 -11040.898} C_VEL
LIN {X 0,Y 403.988,Z 584.741,A -85,B 0,C 180,E1 -11042.525,E2 -11042.525} C_VEL
LIN {X 0,Y 403.541,Z 589.684,A -85,B 0,C 180,E1 -11044.191,E2 -11044.191} C_VEL
LIN {X 0,Y 403.223,Z 593.434,A -85,B 0,C 180,E1 -11045.822,E2 -11045.822} C_VEL
LIN {X 0,Y 402.962,Z 596.401,A -85,B 0,C 180,E1 -11047.572,E2 -11047.572} C_VEL
LIN {X 0,Y 402.777,Z 598.525,A -85,B 0,C 180,E1 -11049.576,E2 -11049.576} C_VEL
LIN {X 0,Y 402.716,Z 599.339,A -85,B 0,C 180,E1 -11051.693,E2 -11051.693} C_VEL
LIN {X 0,Y 402.743,Z 598.694,A -85,B 0,C 180,E1 -11053.788,E2 -11053.788} C_VEL
LIN {X 0,Y 402.84,Z 596.596,A -85,B 0,C 180,E1 -11055.864,E2 -11055.864} C_VEL
LIN {X 0,Y 403.107,Z 593.047,A -85,B 0,C 180,E1 -11057.925,E2 -11057.925} C_VEL
LIN {X 0,Y 403.366,Z 589.423,A -85,B 0,C 180,E1 -11059.46,E2 -11059.46} C_VEL
LIN {X 0,Y 403.694,Z 584.832,A -85,B 0,C 180,E1 -11060.987,E2 -11060.987} C_VEL
LIN {X 0,Y 404.181,Z 578.678,A -85,B 0,C 180,E1 -11062.645,E2 -11062.645} C_VEL
LIN {X 0,Y 404.813,Z 571.27,A -85,B 0,C 180,E1 -11064.272,E2 -11064.272} C_VEL
LIN {X 0,Y 405.587,Z 562.534,A -85,B 0,C 180,E1 -11065.847,E2 -11065.847} C_VEL
LIN {X 0,Y 405.272,Z 558.7,A -85,B 0,C 180,E1 -11066.483,E2 -11066.483} C_VEL
LIN {X 0,Y 403.066,Z 552.286,A -85,B 0,C 180,E1 -11067.512,E2 -11067.512} C_VEL
LIN {X 0,Y 400.941,Z 545.411,A -85,B 0,C 180,E1 -11068.482,E2 -11068.482} C_VEL
LIN {X 0,Y 400.743,Z 540.858,A -85,B 0,C 180,E1 -11069.018,E2 -11069.018} C_VEL
LIN {X 0,Y 401.75,Z 528.375,A -85,B 0,C 180,E1 -11070.251,E2 -11070.251} C_VEL
LIN {X 0,Y 402.801,Z 515.662,A -85,B 0,C 180,E1 -11071.251,E2 -11071.251} C_VEL
LIN {X 0,Y 403.713,Z 502.506,A -85,B 0,C 180,E1 -11072.059,E2 -11072.059} C_VEL
LIN {X 0,Y 404.306,Z 488.434,A -85,B 0,C 180,E1 -11072.71,E2 -11072.71} C_VEL
LIN {X 0,Y 404.819,Z 474.449,A -85,B 0,C 180,E1 -11073.142,E2 -11073.142} C_VEL
LIN {X 0,Y 406.609,Z 363.595,A -85,B 0,C 180,E1 -11075.147,E2 -11075.147} C_VEL
LIN {X 0,Y 403.889,Z 351.912,A -85,B 0,C 180,E1 -11075.514,E2 -11075.514} C_VEL
LIN {X 0,Y 399.122,Z 338.575,A -85,B 0,C 180,E1 -11076.045,E2 -11076.045} C_VEL
LIN {X 0,Y 397.287,Z 329.627,A -85,B 0,C 180,E1 -11078.201,E2 -11078.201} C_VEL
LIN {X 0,Y 397.195,Z 329.637,A -85,B 0,C 180,E1 -11081.224,E2 -11081.224} C_VEL
LIN {X 0,Y 397.173,Z 329.632,A -85,B 0,C 180,E1 -11084.344,E2 -11084.344} C_VEL
LIN {X 0,Y 397.143,Z 329.64,A -85,B 0,C 180,E1 -11087.509,E2 -11087.509} C_VEL
LIN {X 0,Y 397.101,Z 329.644,A -85,B 0,C 180,E1 -11090.731,E2 -11090.731} C_VEL
LIN {X 0,Y 397.105,Z 329.641,A -85,B 0,C 180,E1 -11094.021,E2 -11094.021} C_VEL
LIN {X 0,Y 397.064,Z 329.649,A -85,B 0,C 180,E1 -11097.401,E2 -11097.401} C_VEL
LIN {X 0,Y 397.095,Z 329.642,A -85,B 0,C 180,E1 -11099.863,E2 -11099.863} C_VEL
LIN {X 0,Y 397.109,Z 329.644,A -85,B 0,C 180,E1 -11103.274,E2 -11103.274} C_VEL
LIN {X 0,Y 397.092,Z 329.648,A -85,B 0,C 180,E1 -11106.996,E2 -11106.996} C_VEL
LIN {X 0,Y 397.054,Z 329.65,A -85,B 0,C 180,E1 -11110.438,E2 -11110.438} C_VEL
LIN {X 0,Y 397.086,Z 329.643,A -85,B 0,C 180,E1 -11113.651,E2 -11113.651} C_VEL
LIN {X 0,Y 397.09,Z 329.647,A -85,B 0,C 180,E1 -11116.524,E2 -11116.524} C_VEL
LIN {X 0,Y 397.084,Z 329.648,A -85,B 0,C 180,E1 -11120.42,E2 -11120.42} C_VEL
LIN {X 0,Y 397.092,Z 329.645,A -85,B 0,C 180,E1 -11123.005,E2 -11123.005} C_VEL
LIN {X 0,Y 397.098,Z 329.646,A -85,B 0,C 180,E1 -11126.287,E2 -11126.287} C_VEL
LIN {X 0,Y 397.077,Z 329.646,A -85,B 0,C 180,E1 -11129.118,E2 -11129.118} C_VEL
LIN {X 0,Y 397.062,Z 329.651,A -85,B 0,C 180,E1 -11132.252,E2 -11132.252} C_VEL
LIN {X 0,Y 397.104,Z 329.643,A -85,B 0,C 180,E1 -11134.865,E2 -11134.865} C_VEL
LIN {X 0,Y 397.094,Z 329.647,A -85,B 0,C 180,E1 -11138.182,E2 -11138.182} C_VEL
LIN {X 0,Y 397.152,Z 329.635,A -85,B 0,C 180,E1 -11141.427,E2 -11141.427} C_VEL
LIN {X 0,Y 397.127,Z 329.641,A -85,B 0,C 180,E1 -11144.606,E2 -11144.606} C_VEL
LIN {X 0,Y 397.221,Z 329.629,A -85,B 0,C 180,E1 -11147.742,E2 -11147.742} C_VEL
LIN {X 0,Y 397.238,Z 329.625,A -85,B 0,C 180,E1 -11150.838,E2 -11150.838} C_VEL
LIN {X 0,Y 397.336,Z 329.617,A -85,B 0,C 180,E1 -11153.908,E2 -11153.908} C_VEL
LIN {X 0,Y 397.45,Z 329.605,A -85,B 0,C 180,E1 -11157.974,E2 -11157.974} C_VEL
LIN {X 0,Y 397.575,Z 329.59,A -85,B 0,C 180,E1 -11160,E2 -11160} C_VEL
LIN {X 0,Y 397.34,Z 329.612,A -85,B 0,C 180,E1 -11163.042,E2 -11163.042} C_VEL
LIN {X 0,Y 397.359,Z 329.614,A -85,B 0,C 180,E1 -11166.092,E2 -11166.092} C_VEL
LIN {X 0,Y 397.246,Z 329.624,A -85,B 0,C 180,E1 -11169.162,E2 -11169.162} C_VEL
LIN {X 0,Y 397.223,Z 329.628,A -85,B 0,C 180,E1 -11172.258,E2 -11172.258} C_VEL
LIN {X 0,Y 397.183,Z 329.634,A -85,B 0,C 180,E1 -11175.392,E2 -11175.392} C_VEL
LIN {X 0,Y 397.166,Z 329.633,A -85,B 0,C 180,E1 -11178.574,E2 -11178.574} C_VEL
LIN {X 0,Y 397.113,Z 329.645,A -85,B 0,C 180,E1 -11181.818,E2 -11181.818} C_VEL
LIN {X 0,Y 397.157,Z 329.641,A -85,B 0,C 180,E1 -11185.512,E2 -11185.512} C_VEL
LIN {X 0,Y 397.126,Z 329.638,A -85,B 0,C 180,E1 -11188.544,E2 -11188.544} C_VEL
LIN {X 0,Y 397.082,Z 329.645,A -85,B 0,C 180,E1 -11192.072,E2 -11192.072} C_VEL
LIN {X 0,Y 397.123,Z 329.645,A -85,B 0,C 180,E1 -11195.503,E2 -11195.503} C_VEL
LIN {X 0,Y 397.135,Z 329.639,A -85,B 0,C 180,E1 -11198.861,E2 -11198.861} C_VEL
LIN {X 0,Y 397.075,Z 329.645,A -85,B 0,C 180,E1 -11202.267,E2 -11202.267} C_VEL
LIN {X 0,Y 397.094,Z 329.647,A -85,B 0,C 180,E1 -11205.068,E2 -11205.068} C_VEL
LIN {X 0,Y 397.07,Z 329.646,A -85,B 0,C 180,E1 -11208.021,E2 -11208.021} C_VEL
LIN {X 0,Y 397.134,Z 329.645,A -85,B 0,C 180,E1 -11211.138,E2 -11211.138} C_VEL
LIN {X 0,Y 397.123,Z 329.64,A -85,B 0,C 180,E1 -11214.496,E2 -11214.496} C_VEL
LIN {X 0,Y 397.082,Z 329.649,A -85,B 0,C 180,E1 -11217.928,E2 -11217.928} C_VEL
LIN {X 0,Y 397.117,Z 329.74,A -85,B 0,C 180,E1 -11218.935,E2 -11218.935} C_VEL
LIN {X 0,Y 400.436,Z 344.361,A -85,B 0,C 180,E1 -11221.998,E2 -11221.998} C_VEL
LIN {X 0,Y 401.768,Z 351.031,A -85,B 0,C 180,E1 -11223.346,E2 -11223.346} C_VEL
LIN {X 0,Y 401.053,Z 361.832,A -85,B 0,C 180,E1 -11225.342,E2 -11225.342} C_VEL
LIN {X 0,Y 400.766,Z 365.787,A -85,B 0,C 180,E1 -11226.066,E2 -11226.066} C_VEL
LIN {X 0,Y 406.272,Z 399.357,A -85,B 0,C 180,E1 -11226.995,E2 -11226.995} C_VEL
LIN {X 0,Y 404.532,Z 504.53,A -85,B 0,C 180,E1 -11228.902,E2 -11228.902} C_VEL
LIN {X 0,Y 403.896,Z 519.043,A -85,B 0,C 180,E1 -11229.367,E2 -11229.367} C_VEL
LIN {X 0,Y 403.014,Z 533.102,A -85,B 0,C 180,E1 -11230.026,E2 -11230.026} C_VEL
LIN {X 0,Y 402.175,Z 545.434,A -85,B 0,C 180,E1 -11230.797,E2 -11230.797} C_VEL
LIN {X 0,Y 401.15,Z 557.552,A -85,B 0,C 180,E1 -11231.749,E2 -11231.749} C_VEL
LIN {X 0,Y 400.046,Z 569.269,A -85,B 0,C 180,E1 -11232.886,E2 -11232.886} C_VEL
LIN {X 0,Y 399.031,Z 579.999,A -85,B 0,C 180,E1 -11234.157,E2 -11234.157} C_VEL
LIN {X 0,Y 398.102,Z 590.64,A -85,B 0,C 180,E1 -11235.69,E2 -11235.69} C_VEL
LIN {X 0,Y 397.409,Z 599.415,A -85,B 0,C 180,E1 -11237.228,E2 -11237.228} C_VEL
LIN {X 0,Y 396.66,Z 607.809,A -85,B 0,C 180,E1 -11239.019,E2 -11239.019} C_VEL
LIN {X 0,Y 396.212,Z 614.543,A -85,B 0,C 180,E1 -11240.813,E2 -11240.813} C_VEL
LIN {X 0,Y 395.91,Z 620.508,A -85,B 0,C 180,E1 -11242.861,E2 -11242.861} C_VEL
LIN {X 0,Y 395.813,Z 624.868,A -85,B 0,C 180,E1 -11244.906,E2 -11244.906} C_VEL
LIN {X 0,Y 395.755,Z 627.756,A -85,B 0,C 180,E1 -11246.945,E2 -11246.945} C_VEL
LIN {X 0,Y 395.839,Z 628.681,A -85,B 0,C 180,E1 -11247.964,E2 -11247.964} C_VEL
LIN {X 0,Y 395.796,Z 629.501,A -85,B 0,C 180,E1 -11249.999,E2 -11249.999} C_VEL
LIN {X 0,Y 395.802,Z 628.978,A -85,B 0,C 180,E1 -11252.034,E2 -11252.034} C_VEL
LIN {X 0,Y 395.763,Z 627.11,A -85,B 0,C 180,E1 -11254.072,E2 -11254.072} C_VEL
LIN {X 0,Y 395.861,Z 623.857,A -85,B 0,C 180,E1 -11256.114,E2 -11256.114} C_VEL
LIN {X 0,Y 395.998,Z 620.414,A -85,B 0,C 180,E1 -11257.648,E2 -11257.648} C_VEL
LIN {X 0,Y 396.359,Z 614.487,A -85,B 0,C 180,E1 -11259.697,E2 -11259.697} C_VEL
LIN {X 0,Y 396.97,Z 607.846,A -85,B 0,C 180,E1 -11261.487,E2 -11261.487} C_VEL
LIN {X 0,Y 397.735,Z 599.627,A -85,B 0,C 180,E1 -11263.279,E2 -11263.279} C_VEL
LIN {X 0,Y 398.613,Z 591.064,A -85,B 0,C 180,E1 -11264.811,E2 -11264.811} C_VEL
LIN {X 0,Y 399.744,Z 580.722,A -85,B 0,C 180,E1 -11266.337,E2 -11266.337} C_VEL
LIN {X 0,Y 401.113,Z 569.19,A -85,B 0,C 180,E1 -11267.723,E2 -11267.723} C_VEL
LIN {X 0,Y 402.318,Z 557.722,A -85,B 0,C 180,E1 -11268.854,E2 -11268.854} C_VEL
LIN {X 0,Y 403.634,Z 544.369,A -85,B 0,C 180,E1 -11269.908,E2 -11269.908} C_VEL
LIN {X 0,Y 404.652,Z 531.154,A -85,B 0,C 180,E1 -11270.723,E2 -11270.723} C_VEL
LIN {X 0,Y 405.666,Z 516.964,A -85,B 0,C 180,E1 -11271.367,E2 -11271.367} C_VEL
LIN {X 0,Y 406.418,Z 502.99,A -85,B 0,C 180,E1 -11271.791,E2 -11271.791} C_VEL
LIN {X 0,Y 408.274,Z 398.861,A -85,B 0,C 180,E1 -11273.714,E2 -11273.714} C_VEL
LIN {X 0,Y 403.966,Z 374.716,A -85,B 0,C 180,E1 -11274.5,E2 -11274.5} C_VEL
LIN {X 0,Y 401.883,Z 364.969,A -85,B 0,C 180,E1 -11274.884,E2 -11274.884} C_VEL
LIN {X 0,Y 402.826,Z 355.429,A -85,B 0,C 180,E1 -11276.695,E2 -11276.695} C_VEL
LIN {X 0,Y 401.982,Z 349.819,A -85,B 0,C 180,E1 -11277.882,E2 -11277.882} C_VEL
LIN {X 0,Y 399.389,Z 338.473,A -85,B 0,C 180,E1 -11280.43,E2 -11280.43} C_VEL
LIN {X 0,Y 397.089,Z 329.649,A -85,B 0,C 180,E1 -11282.557,E2 -11282.557} C_VEL
LIN {X 0,Y 397.106,Z 329.641,A -85,B 0,C 180,E1 -11285.733,E2 -11285.733} C_VEL
LIN {X 0,Y 397.133,Z 329.636,A -85,B 0,C 180,E1 -11288.862,E2 -11288.862} C_VEL
LIN {X 0,Y 397.11,Z 329.636,A -85,B 0,C 180,E1 -11292.26,E2 -11292.26} C_VEL
LIN {X 0,Y 397.084,Z 329.639,A -85,B 0,C 180,E1 -11295.067,E2 -11295.067} C_VEL
LIN {X 0,Y 397.069,Z 329.649,A -85,B 0,C 180,E1 -11298.019,E2 -11298.019} C_VEL
LIN {X 0,Y 397.126,Z 329.633,A -85,B 0,C 180,E1 -11301.137,E2 -11301.137} C_VEL
LIN {X 0,Y 397.114,Z 329.642,A -85,B 0,C 180,E1 -11304.496,E2 -11304.496} C_VEL
LIN {X 0,Y 397.075,Z 329.645,A -85,B 0,C 180,E1 -11307.928,E2 -11307.928} C_VEL
LIN {X 0,Y 397.12,Z 329.64,A -85,B 0,C 180,E1 -11311.456,E2 -11311.456} C_VEL
LIN {X 0,Y 397.146,Z 329.639,A -85,B 0,C 180,E1 -11314.487,E2 -11314.487} C_VEL
LIN {X 0,Y 397.1,Z 329.643,A -85,B 0,C 180,E1 -11318.181,E2 -11318.181} C_VEL
LIN {X 0,Y 397.155,Z 329.631,A -85,B 0,C 180,E1 -11321.426,E2 -11321.426} C_VEL
LIN {X 0,Y 397.176,Z 329.628,A -85,B 0,C 180,E1 -11324.608,E2 -11324.608} C_VEL
LIN {X 0,Y 397.21,Z 329.633,A -85,B 0,C 180,E1 -11327.741,E2 -11327.741} C_VEL
LIN {X 0,Y 397.386,Z 329.607,A -85,B 0,C 180,E1 -11332.041,E2 -11332.041} C_VEL
LIN {X 0,Y 397.237,Z 329.626,A -85,B 0,C 180,E1 -11334.925,E2 -11334.925} C_VEL
LIN {X 0,Y 397.432,Z 329.602,A -85,B 0,C 180,E1 -11337.973,E2 -11337.973} C_VEL
LIN {X 0,Y 397.436,Z 329.602,A -85,B 0,C 180,E1 -11342.026,E2 -11342.026} C_VEL
LIN {X 0,Y 397.281,Z 329.62,A -85,B 0,C 180,E1 -11346.49,E2 -11346.49} C_VEL
LIN {X 0,Y 397.219,Z 329.626,A -85,B 0,C 180,E1 -11349.162,E2 -11349.162} C_VEL
LIN {X 0,Y 397.208,Z 329.626,A -85,B 0,C 180,E1 -11352.258,E2 -11352.258} C_VEL
LIN {X 0,Y 397.161,Z 329.636,A -85,B 0,C 180,E1 -11355.392,E2 -11355.392} C_VEL
LIN {X 0,Y 397.145,Z 329.638,A -85,B 0,C 180,E1 -11358.574,E2 -11358.574} C_VEL
LIN {X 0,Y 397.086,Z 329.642,A -85,B 0,C 180,E1 -11361.819,E2 -11361.819} C_VEL
LIN {X 0,Y 397.098,Z 329.645,A -85,B 0,C 180,E1 -11365.135,E2 -11365.135} C_VEL
LIN {X 0,Y 397.062,Z 329.639,A -85,B 0,C 180,E1 -11368.548,E2 -11368.548} C_VEL
LIN {X 0,Y 397.072,Z 329.649,A -85,B 0,C 180,E1 -11371.837,E2 -11371.837} C_VEL
LIN {X 0,Y 397.115,Z 329.646,A -85,B 0,C 180,E1 -11374.494,E2 -11374.494} C_VEL
LIN {X 0,Y 397.091,Z 329.649,A -85,B 0,C 180,E1 -11378.276,E2 -11378.276} C_VEL
LIN {X 0,Y 397.08,Z 329.65,A -85,B 0,C 180,E1 -11380.909,E2 -11380.909} C_VEL
LIN {X 0,Y 397.119,Z 329.777,A -85,B 0,C 180,E1 -11384.475,E2 -11384.475} C_VEL
LIN {X 0,Y 399.404,Z 339.345,A -85,B 0,C 180,E1 -11387.01,E2 -11387.01} C_VEL
LIN {X 0,Y 407.436,Z 358.026,A -85,B 0,C 180,E1 -11387.993,E2 -11387.993} C_VEL
LIN {X 0,Y 408.943,Z 364.824,A -85,B 0,C 180,E1 -11388.236,E2 -11388.236} C_VEL
LIN {X 0,Y 406.769,Z 475.135,A -85,B 0,C 180,E1 -11390.264,E2 -11390.264} C_VEL
LIN {X 0,Y 406.211,Z 489.436,A -85,B 0,C 180,E1 -11390.721,E2 -11390.721} C_VEL
LIN {X 0,Y 405.436,Z 502.271,A -85,B 0,C 180,E1 -11391.311,E2 -11391.311} C_VEL
LIN {X 0,Y 404.569,Z 514.896,A -85,B 0,C 180,E1 -11392.084,E2 -11392.084} C_VEL
LIN {X 0,Y 403.386,Z 527.768,A -85,B 0,C 180,E1 -11393.088,E2 -11393.088} C_VEL
LIN {X 0,Y 402.08,Z 540.287,A -85,B 0,C 180,E1 -11394.314,E2 -11394.314} C_VEL
LIN {X 0,Y 400.939,Z 550.714,A -85,B 0,C 180,E1 -11395.569,E2 -11395.569} C_VEL
LIN {X 0,Y 399.82,Z 560.452,A -85,B 0,C 180,E1 -11396.983,E2 -11396.983} C_VEL
LIN {X 0,Y 398.717,Z 570.009,A -85,B 0,C 180,E1 -11398.67,E2 -11398.67} C_VEL
LIN {X 0,Y 397.806,Z 577.775,A -85,B 0,C 180,E1 -11400.353,E2 -11400.353} C_VEL
LIN {X 0,Y 397.023,Z 584.854,A -85,B 0,C 180,E1 -11402.261,E2 -11402.261} C_VEL
LIN {X 0,Y 396.466,Z 590.573,A -85,B 0,C 180,E1 -11404.261,E2 -11404.261} C_VEL
LIN {X 0,Y 396.124,Z 594.211,A -85,B 0,C 180,E1 -11405.918,E2 -11405.918} C_VEL
LIN {X 0,Y 395.907,Z 596.573,A -85,B 0,C 180,E1 -11407.38,E2 -11407.38} C_VEL
LIN {X 0,Y 395.723,Z 598.569,A -85,B 0,C 180,E1 -11409.196,E2 -11409.196} C_VEL
LIN {X 0,Y 395.635,Z 599.566,A -85,B 0,C 180,E1 -11411.353,E2 -11411.353} C_VEL
LIN {X 0,Y 395.661,Z 599.074,A -85,B 0,C 180,E1 -11413.572,E2 -11413.572} C_VEL
LIN {X 0,Y 395.742,Z 597.243,A -85,B 0,C 180,E1 -11415.605,E2 -11415.605} C_VEL
LIN {X 0,Y 396.007,Z 593.905,A -85,B 0,C 180,E1 -11417.705,E2 -11417.705} C_VEL
LIN {X 0,Y 396.319,Z 589.036,A -85,B 0,C 180,E1 -11419.787,E2 -11419.787} C_VEL
LIN {X 0,Y 396.718,Z 584.335,A -85,B 0,C 180,E1 -11421.34,E2 -11421.34} C_VEL
LIN {X 0,Y 397.263,Z 577.513,A -85,B 0,C 180,E1 -11423.143,E2 -11423.143} C_VEL
LIN {X 0,Y 398.065,Z 569.038,A -85,B 0,C 180,E1 -11424.936,E2 -11424.936} C_VEL
LIN {X 0,Y 398.899,Z 560.211,A -85,B 0,C 180,E1 -11426.466,E2 -11426.466} C_VEL
LIN {X 0,Y 399.917,Z 549.528,A -85,B 0,C 180,E1 -11427.987,E2 -11427.987} C_VEL
LIN {X 0,Y 400.743,Z 540.858,A -85,B 0,C 180,E1 -11429.018,E2 -11429.018} C_VEL
LIN {X 0,Y 400.535,Z 536.243,A -85,B 0,C 180,E1 -11429.534,E2 -11429.534} C_VEL
LIN {X 0,Y 398.388,Z 528.571,A -85,B 0,C 180,E1 -11430.379,E2 -11430.379} C_VEL
LIN {X 0,Y 396.256,Z 520.592,A -85,B 0,C 180,E1 -11431.17,E2 -11431.17} C_VEL
LIN {X 0,Y 396.052,Z 515.347,A -85,B 0,C 180,E1 -11431.583,E2 -11431.583} C_VEL
LIN {X 0,Y 396.984,Z 501.919,A -85,B 0,C 180,E1 -11432.411,E2 -11432.411} C_VEL
LIN {X 0,Y 397.606,Z 487.42,A -85,B 0,C 180,E1 -11433.072,E2 -11433.072} C_VEL
LIN {X 0,Y 398.133,Z 473.908,A -85,B 0,C 180,E1 -11433.48,E2 -11433.48} C_VEL
LIN {X 0,Y 399.927,Z 364.363,A -85,B 0,C 180,E1 -11435.493,E2 -11435.493} C_VEL
LIN {X 0,Y 397.605,Z 354.516,A -85,B 0,C 180,E1 -11435.809,E2 -11435.809} C_VEL
LIN {X 0,Y 391.937,Z 338.905,A -85,B 0,C 180,E1 -11436.436,E2 -11436.436} C_VEL
LIN {X 0,Y 390.22,Z 330.505,A -85,B 0,C 180,E1 -11438.481,E2 -11438.481} C_VEL
LIN {X 0,Y 390.144,Z 330.514,A -85,B 0,C 180,E1 -11441.43,E2 -11441.43} C_VEL
LIN {X 0,Y 390.141,Z 330.509,A -85,B 0,C 180,E1 -11444.608,E2 -11444.608} C_VEL
LIN {X 0,Y 390.11,Z 330.513,A -85,B 0,C 180,E1 -11447.835,E2 -11447.835} C_VEL
LIN {X 0,Y 390.054,Z 330.526,A -85,B 0,C 180,E1 -11451.123,E2 -11451.123} C_VEL
LIN {X 0,Y 390.04,Z 330.522,A -85,B 0,C 180,E1 -11454.484,E2 -11454.484} C_VEL
LIN {X 0,Y 390.014,Z 330.524,A -85,B 0,C 180,E1 -11457.998,E2 -11457.998} C_VEL
LIN {X 0,Y 390.016,Z 330.526,A -85,B 0,C 180,E1 -11461.506,E2 -11461.506} C_VEL
LIN {X 0,Y 390.067,Z 330.521,A -85,B 0,C 180,E1 -11465.21,E2 -11465.21} C_VEL
LIN {X 0,Y 390.056,Z 330.523,A -85,B 0,C 180,E1 -11469.097,E2 -11469.097} C_VEL
LIN {X 0,Y 390.029,Z 330.525,A -85,B 0,C 180,E1 -11472.373,E2 -11472.373} C_VEL
LIN {X 0,Y 390.04,Z 330.522,A -85,B 0,C 180,E1 -11475.354,E2 -11475.354} C_VEL
LIN {X 0,Y 390.014,Z 330.526,A -85,B 0,C 180,E1 -11478.185,E2 -11478.185} C_VEL
LIN {X 0,Y 390.054,Z 330.523,A -85,B 0,C 180,E1 -11480.904,E2 -11480.904} C_VEL
LIN {X 0,Y 390.08,Z 330.52,A -85,B 0,C 180,E1 -11484.793,E2 -11484.793} C_VEL
LIN {X 0,Y 390.023,Z 330.53,A -85,B 0,C 180,E1 -11488.496,E2 -11488.496} C_VEL
LIN {X 0,Y 390.016,Z 330.526,A -85,B 0,C 180,E1 -11492.004,E2 -11492.004} C_VEL
LIN {X 0,Y 390.043,Z 330.521,A -85,B 0,C 180,E1 -11495.517,E2 -11495.517} C_VEL
LIN {X 0,Y 390.054,Z 330.521,A -85,B 0,C 180,E1 -11498.878,E2 -11498.878} C_VEL
LIN {X 0,Y 390.105,Z 330.518,A -85,B 0,C 180,E1 -11502.166,E2 -11502.166} C_VEL
LIN {X 0,Y 390.094,Z 330.514,A -85,B 0,C 180,E1 -11505.391,E2 -11505.391} C_VEL
LIN {X 0,Y 390.173,Z 330.505,A -85,B 0,C 180,E1 -11507.517,E2 -11507.517} C_VEL
LIN {X 0,Y 390.195,Z 330.503,A -85,B 0,C 180,E1 -11510.671,E2 -11510.671} C_VEL
LIN {X 0,Y 390.29,Z 330.493,A -85,B 0,C 180,E1 -11513.798,E2 -11513.798} C_VEL
LIN {X 0,Y 390.417,Z 330.48,A -85,B 0,C 180,E1 -11517.937,E2 -11517.937} C_VEL
LIN {X 0,Y 390.545,Z 330.465,A -85,B 0,C 180,E1 -11520,E2 -11520} C_VEL
LIN {X 0,Y 390.276,Z 330.492,A -85,B 0,C 180,E1 -11523.097,E2 -11523.097} C_VEL
LIN {X 0,Y 390.311,Z 330.491,A -85,B 0,C 180,E1 -11526.203,E2 -11526.203} C_VEL
LIN {X 0,Y 390.201,Z 330.503,A -85,B 0,C 180,E1 -11529.329,E2 -11529.329} C_VEL
LIN {X 0,Y 390.174,Z 330.505,A -85,B 0,C 180,E1 -11532.483,E2 -11532.483} C_VEL
LIN {X 0,Y 390.143,Z 330.515,A -85,B 0,C 180,E1 -11535.677,E2 -11535.677} C_VEL
LIN {X 0,Y 390.11,Z 330.513,A -85,B 0,C 180,E1 -11538.922,E2 -11538.922} C_VEL
LIN {X 0,Y 390.051,Z 330.521,A -85,B 0,C 180,E1 -11542.234,E2 -11542.234} C_VEL
LIN {X 0,Y 390.123,Z 330.515,A -85,B 0,C 180,E1 -11545.743,E2 -11545.743} C_VEL
LIN {X 0,Y 390.063,Z 330.521,A -85,B 0,C 180,E1 -11549.11,E2 -11549.11} C_VEL
LIN {X 0,Y 390.047,Z 330.521,A -85,B 0,C 180,E1 -11552.721,E2 -11552.721} C_VEL
LIN {X 0,Y 390.06,Z 330.521,A -85,B 0,C 180,E1 -11555.825,E2 -11555.825} C_VEL
LIN {X 0,Y 390.074,Z 330.522,A -85,B 0,C 180,E1 -11559.218,E2 -11559.218} C_VEL
LIN {X 0,Y 390.048,Z 330.52,A -85,B 0,C 180,E1 -11562.374,E2 -11562.374} C_VEL
LIN {X 0,Y 390.05,Z 330.525,A -85,B 0,C 180,E1 -11565.354,E2 -11565.354} C_VEL
LIN {X 0,Y 390.035,Z 330.522,A -85,B 0,C 180,E1 -11568.186,E2 -11568.186} C_VEL
LIN {X 0,Y 390.094,Z 330.519,A -85,B 0,C 180,E1 -11570.907,E2 -11570.907} C_VEL
LIN {X 0,Y 390.089,Z 330.519,A -85,B 0,C 180,E1 -11574.793,E2 -11574.793} C_VEL
LIN {X 0,Y 390.076,Z 330.581,A -85,B 0,C 180,E1 -11578.612,E2 -11578.612} C_VEL
LIN {X 0,Y 393.731,Z 346.745,A -85,B 0,C 180,E1 -11582.059,E2 -11582.059} C_VEL
LIN {X 0,Y 394.884,Z 353.06,A -85,B 0,C 180,E1 -11583.351,E2 -11583.351} C_VEL
LIN {X 0,Y 393.901,Z 365.475,A -85,B 0,C 180,E1 -11585.675,E2 -11585.675} C_VEL
LIN {X 0,Y 399.603,Z 400.621,A -85,B 0,C 180,E1 -11586.671,E2 -11586.671} C_VEL
LIN {X 0,Y 397.841,Z 503.613,A -85,B 0,C 180,E1 -11588.564,E2 -11588.564} C_VEL
LIN {X 0,Y 397.172,Z 518.346,A -85,B 0,C 180,E1 -11589.036,E2 -11589.036} C_VEL
LIN {X 0,Y 396.282,Z 532.404,A -85,B 0,C 180,E1 -11589.699,E2 -11589.699} C_VEL
LIN {X 0,Y 395.295,Z 545.992,A -85,B 0,C 180,E1 -11590.565,E2 -11590.565} C_VEL
LIN {X 0,Y 394.216,Z 558.163,A -85,B 0,C 180,E1 -11591.551,E2 -11591.551} C_VEL
LIN {X 0,Y 393.084,Z 569.726,A -85,B 0,C 180,E1 -11592.707,E2 -11592.707} C_VEL
LIN {X 0,Y 392.137,Z 579.353,A -85,B 0,C 180,E1 -11593.87,E2 -11593.87} C_VEL
LIN {X 0,Y 391.149,Z 590.067,A -85,B 0,C 180,E1 -11595.43,E2 -11595.43} C_VEL
LIN {X 0,Y 390.435,Z 598.904,A -85,B 0,C 180,E1 -11596.996,E2 -11596.996} C_VEL
LIN {X 0,Y 389.645,Z 607.357,A -85,B 0,C 180,E1 -11598.819,E2 -11598.819} C_VEL
LIN {X 0,Y 389.138,Z 614.138,A -85,B 0,C 180,E1 -11600.645,E2 -11600.645} C_VEL
LIN {X 0,Y 388.83,Z 620.138,A -85,B 0,C 180,E1 -11602.73,E2 -11602.73} C_VEL
LIN {X 0,Y 388.716,Z 624.528,A -85,B 0,C 180,E1 -11604.812,E2 -11604.812} C_VEL
LIN {X 0,Y 388.659,Z 627.442,A -85,B 0,C 180,E1 -11606.889,E2 -11606.889} C_VEL
LIN {X 0,Y 388.74,Z 628.972,A -85,B 0,C 180,E1 -11608.963,E2 -11608.963} C_VEL
LIN {X 0,Y 388.738,Z 629.145,A -85,B 0,C 180,E1 -11611.035,E2 -11611.035} C_VEL
LIN {X 0,Y 388.634,Z 627.972,A -85,B 0,C 180,E1 -11613.109,E2 -11613.109} C_VEL
LIN {X 0,Y 388.703,Z 625.451,A -85,B 0,C 180,E1 -11615.186,E2 -11615.186} C_VEL
LIN {X 0,Y 388.906,Z 621.504,A -85,B 0,C 180,E1 -11617.266,E2 -11617.266} C_VEL
LIN {X 0,Y 389.203,Z 615.989,A -85,B 0,C 180,E1 -11619.352,E2 -11619.352} C_VEL
LIN {X 0,Y 389.711,Z 609.785,A -85,B 0,C 180,E1 -11621.177,E2 -11621.177} C_VEL
LIN {X 0,Y 390.474,Z 602.072,A -85,B 0,C 180,E1 -11623.001,E2 -11623.001} C_VEL
LIN {X 0,Y 391.536,Z 592.565,A -85,B 0,C 180,E1 -11624.819,E2 -11624.819} C_VEL
LIN {X 0,Y 392.66,Z 582.633,A -85,B 0,C 180,E1 -11626.373,E2 -11626.373} C_VEL
LIN {X 0,Y 394.079,Z 571.621,A -85,B 0,C 180,E1 -11627.782,E2 -11627.782} C_VEL
LIN {X 0,Y 395.463,Z 559.399,A -85,B 0,C 180,E1 -11629.059,E2 -11629.059} C_VEL
LIN {X 0,Y 396.764,Z 547.117,A -85,B 0,C 180,E1 -11630.088,E2 -11630.088} C_VEL
LIN {X 0,Y 397.873,Z 534.021,A -85,B 0,C 180,E1 -11630.957,E2 -11630.957} C_VEL
LIN {X 0,Y 398.992,Z 520.184,A -85,B 0,C 180,E1 -11631.641,E2 -11631.641} C_VEL
LIN {X 0,Y 399.837,Z 505.772,A -85,B 0,C 180,E1 -11632.135,E2 -11632.135} C_VEL
LIN {X 0,Y 400.342,Z 484.225,A -85,B 0,C 180,E1 -11632.581,E2 -11632.581} C_VEL
LIN {X 0,Y 401.926,Z 400.126,A -85,B 0,C 180,E1 -11634.141,E2 -11634.141} C_VEL
LIN {X 0,Y 397.922,Z 377.112,A -85,B 0,C 180,E1 -11634.904,E2 -11634.904} C_VEL
LIN {X 0,Y 395.21,Z 364.728,A -85,B 0,C 180,E1 -11635.39,E2 -11635.39} C_VEL
LIN {X 0,Y 396.039,Z 357.082,A -85,B 0,C 180,E1 -11636.869,E2 -11636.869} C_VEL
LIN {X 0,Y 395.124,Z 351.318,A -85,B 0,C 180,E1 -11638.121,E2 -11638.121} C_VEL
LIN {X 0,Y 392.301,Z 339.203,A -85,B 0,C 180,E1 -11640.913,E2 -11640.913} C_VEL
LIN {X 0,Y 390.065,Z 330.523,A -85,B 0,C 180,E1 -11643.064,E2 -11643.064} C_VEL
LIN {X 0,Y 390.057,Z 330.518,A -85,B 0,C 180,E1 -11646.482,E2 -11646.482} C_VEL
LIN {X 0,Y 390.07,Z 330.517,A -85,B 0,C 180,E1 -11649.218,E2 -11649.218} C_VEL
LIN {X 0,Y 390.076,Z 330.512,A -85,B 0,C 180,E1 -11652.379,E2 -11652.379} C_VEL
LIN {X 0,Y 390.052,Z 330.511,A -85,B 0,C 180,E1 -11656.112,E2 -11656.112} C_VEL
LIN {X 0,Y 390.056,Z 330.514,A -85,B 0,C 180,E1 -11659.56,E2 -11659.56} C_VEL
LIN {X 0,Y 390.04,Z 330.525,A -85,B 0,C 180,E1 -11662.448,E2 -11662.448} C_VEL
LIN {X 0,Y 390.062,Z 330.523,A -85,B 0,C 180,E1 -11665.974,E2 -11665.974} C_VEL
LIN {X 0,Y 390.046,Z 330.522,A -85,B 0,C 180,E1 -11669.867,E2 -11669.867} C_VEL
LIN {X 0,Y 390.107,Z 330.51,A -85,B 0,C 180,E1 -11673.231,E2 -11673.231} C_VEL
LIN {X 0,Y 390.069,Z 330.514,A -85,B 0,C 180,E1 -11676.76,E2 -11676.76} C_VEL
LIN {X 0,Y 390.096,Z 330.517,A -85,B 0,C 180,E1 -11679.982,E2 -11679.982} C_VEL
LIN {X 0,Y 390.134,Z 330.512,A -85,B 0,C 180,E1 -11683.248,E2 -11683.248} C_VEL
LIN {X 0,Y 390.186,Z 330.506,A -85,B 0,C 180,E1 -11686.561,E2 -11686.561} C_VEL
LIN {X 0,Y 390.196,Z 330.504,A -85,B 0,C 180,E1 -11690.671,E2 -11690.671} C_VEL
LIN {X 0,Y 390.308,Z 330.483,A -85,B 0,C 180,E1 -11692.759,E2 -11692.759} C_VEL
LIN {X 0,Y 390.21,Z 330.502,A -85,B 0,C 180,E1 -11694.833,E2 -11694.833} C_VEL
LIN {X 0,Y 390.4,Z 330.477,A -85,B 0,C 180,E1 -11697.936,E2 -11697.936} C_VEL
LIN {X 0,Y 390.403,Z 330.478,A -85,B 0,C 180,E1 -11702.063,E2 -11702.063} C_VEL
LIN {X 0,Y 390.241,Z 330.497,A -85,B 0,C 180,E1 -11706.481,E2 -11706.481} C_VEL
LIN {X 0,Y 390.177,Z 330.503,A -85,B 0,C 180,E1 -11709.329,E2 -11709.329} C_VEL
LIN {X 0,Y 390.16,Z 330.503,A -85,B 0,C 180,E1 -11712.483,E2 -11712.483} C_VEL
LIN {X 0,Y 390.123,Z 330.51,A -85,B 0,C 180,E1 -11715.677,E2 -11715.677} C_VEL
LIN {X 0,Y 390.091,Z 330.517,A -85,B 0,C 180,E1 -11718.922,E2 -11718.922} C_VEL
LIN {X 0,Y 390.029,Z 330.52,A -85,B 0,C 180,E1 -11722.234,E2 -11722.234} C_VEL
LIN {X 0,Y 390.04,Z 330.527,A -85,B 0,C 180,E1 -11725.722,E2 -11725.722} C_VEL
LIN {X 0,Y 390.019,Z 330.518,A -85,B 0,C 180,E1 -11729.112,E2 -11729.112} C_VEL
LIN {X 0,Y 390.033,Z 330.52,A -85,B 0,C 180,E1 -11732.722,E2 -11732.722} C_VEL
LIN {X 0,Y 390.046,Z 330.524,A -85,B 0,C 180,E1 -11735.826,E2 -11735.826} C_VEL
LIN {X 0,Y 390.058,Z 330.518,A -85,B 0,C 180,E1 -11739.218,E2 -11739.218} C_VEL
LIN {X 0,Y 390.033,Z 330.522,A -85,B 0,C 180,E1 -11742.375,E2 -11742.375} C_VEL
LIN {X 0,Y 390.077,Z 330.704,A -85,B 0,C 180,E1 -11744.008,E2 -11744.008} C_VEL
LIN {X 0,Y 392.24,Z 339.597,A -85,B 0,C 180,E1 -11746.43,E2 -11746.43} C_VEL
LIN {X 0,Y 400.823,Z 358.993,A -85,B 0,C 180,E1 -11747.52,E2 -11747.52} C_VEL
LIN {X 0,Y 402.184,Z 364.067,A -85,B 0,C 180,E1 -11747.726,E2 -11747.726} C_VEL
LIN {X 0,Y 402.607,Z 366.142,A -85,B 0,C 180,E1 -11747.799,E2 -11747.799} C_VEL
LIN {X 0,Y 400.318,Z 476.305,A -85,B 0,C 180,E1 -11749.863,E2 -11749.863} C_VEL
LIN {X 0,Y 399.707,Z 490.238,A -85,B 0,C 180,E1 -11750.323,E2 -11750.323} C_VEL
LIN {X 0,Y 398.888,Z 503.812,A -85,B 0,C 180,E1 -11750.975,E2 -11750.975} C_VEL
LIN {X 0,Y 397.853,Z 516.913,A -85,B 0,C 180,E1 -11751.812,E2 -11751.812} C_VEL
LIN {X 0,Y 396.607,Z 529.986,A -85,B 0,C 180,E1 -11752.883,E2 -11752.883} C_VEL
LIN {X 0,Y 395.286,Z 541.684,A -85,B 0,C 180,E1 -11754.077,E2 -11754.077} C_VEL
LIN {X 0,Y 393.984,Z 553.037,A -85,B 0,C 180,E1 -11755.504,E2 -11755.504} C_VEL
LIN {X 0,Y 392.671,Z 563.622,A -85,B 0,C 180,E1 -11757.148,E2 -11757.148} C_VEL
LIN {X 0,Y 391.505,Z 572.835,A -85,B 0,C 180,E1 -11758.91,E2 -11758.91} C_VEL
LIN {X 0,Y 390.606,Z 580.194,A -85,B 0,C 180,E1 -11760.641,E2 -11760.641} C_VEL
LIN {X 0,Y 389.841,Z 586.953,A -85,B 0,C 180,E1 -11762.633,E2 -11762.633} C_VEL
LIN {X 0,Y 389.331,Z 591.849,A -85,B 0,C 180,E1 -11764.497,E2 -11764.497} C_VEL
LIN {X 0,Y 388.931,Z 595.874,A -85,B 0,C 180,E1 -11766.577,E2 -11766.577} C_VEL
LIN {X 0,Y 388.776,Z 597.452,A -85,B 0,C 180,E1 -11767.691,E2 -11767.691} C_VEL
LIN {X 0,Y 388.61,Z 599.39,A -85,B 0,C 180,E1 -11769.904,E2 -11769.904} C_VEL
LIN {X 0,Y 388.512,Z 599.839,A -85,B 0,C 180,E1 -11772.091,E2 -11772.091} C_VEL
LIN {X 0,Y 388.582,Z 598.85,A -85,B 0,C 180,E1 -11774.26,E2 -11774.26} C_VEL
LIN {X 0,Y 388.704,Z 596.446,A -85,B 0,C 180,E1 -11776.407,E2 -11776.407} C_VEL
LIN {X 0,Y 388.958,Z 593.67,A -85,B 0,C 180,E1 -11778.008,E2 -11778.008} C_VEL
LIN {X 0,Y 389.2,Z 590.076,A -85,B 0,C 180,E1 -11779.598,E2 -11779.598} C_VEL
LIN {X 0,Y 389.581,Z 585.496,A -85,B 0,C 180,E1 -11781.181,E2 -11781.181} C_VEL
LIN {X 0,Y 390.162,Z 578.906,A -85,B 0,C 180,E1 -11783.017,E2 -11783.017} C_VEL
LIN {X 0,Y 390.951,Z 570.736,A -85,B 0,C 180,E1 -11784.844,E2 -11784.844} C_VEL
LIN {X 0,Y 391.747,Z 562.205,A -85,B 0,C 180,E1 -11786.401,E2 -11786.401} C_VEL
LIN {X 0,Y 392.806,Z 551.856,A -85,B 0,C 180,E1 -11787.95,E2 -11787.95} C_VEL
LIN {X 0,Y 393.911,Z 540.857,A -85,B 0,C 180,E1 -11789.3,E2 -11789.3} C_VEL
LIN {X 0,Y 394.897,Z 528.806,A -85,B 0,C 180,E1 -11790.511,E2 -11790.511} C_VEL
LIN {X 0,Y 396.052,Z 515.347,A -85,B 0,C 180,E1 -11791.583,E2 -11791.583} C_VEL
LIN {X 0,Y 395.795,Z 510.072,A -85,B 0,C 180,E1 -11791.974,E2 -11791.974} C_VEL
LIN {X 0,Y 393.453,Z 501.463,A -85,B 0,C 180,E1 -11792.622,E2 -11792.622} C_VEL
LIN {X 0,Y 391.146,Z 492.607,A -85,B 0,C 180,E1 -11793.179,E2 -11793.179} C_VEL
LIN {X 0,Y 390.921,Z 486.96,A -85,B 0,C 180,E1 -11793.421,E2 -11793.421} C_VEL
LIN {X 0,Y 391.454,Z 473.263,A -85,B 0,C 180,E1 -11793.829,E2 -11793.829} C_VEL
LIN {X 0,Y 393.286,Z 365.489,A -85,B 0,C 180,E1 -11795.837,E2 -11795.837} C_VEL
LIN {X 0,Y 391.173,Z 356.702,A -85,B 0,C 180,E1 -11796.129,E2 -11796.129} C_VEL
LIN {X 0,Y 384.767,Z 339.005,A -85,B 0,C 180,E1 -11796.885,E2 -11796.885} C_VEL
LIN {X 0,Y 383.172,Z 331.382,A -85,B 0,C 180,E1 -11798.837,E2 -11798.837} C_VEL
LIN {X 0,Y 383.134,Z 331.383,A -85,B 0,C 180,E1 -11802.717,E2 -11802.717} C_VEL
LIN {X 0,Y 383.078,Z 331.389,A -85,B 0,C 180,E1 -11805.974,E2 -11805.974} C_VEL
LIN {X 0,Y 383.057,Z 331.397,A -85,B 0,C 180,E1 -11809.285,E2 -11809.285} C_VEL
LIN {X 0,Y 382.988,Z 331.402,A -85,B 0,C 180,E1 -11812.667,E2 -11812.667} C_VEL
LIN {X 0,Y 382.981,Z 331.4,A -85,B 0,C 180,E1 -11816.131,E2 -11816.131} C_VEL
LIN {X 0,Y 382.973,Z 331.402,A -85,B 0,C 180,E1 -11819.702,E2 -11819.702} C_VEL
LIN {X 0,Y 382.997,Z 331.4,A -85,B 0,C 180,E1 -11823.402,E2 -11823.402} C_VEL
LIN {X 0,Y 383.02,Z 331.396,A -85,B 0,C 180,E1 -11826.163,E2 -11826.163} C_VEL
LIN {X 0,Y 382.984,Z 331.4,A -85,B 0,C 180,E1 -11829.582,E2 -11829.582} C_VEL
LIN {X 0,Y 383.006,Z 331.404,A -85,B 0,C 180,E1 -11832.779,E2 -11832.779} C_VEL
LIN {X 0,Y 382.989,Z 331.399,A -85,B 0,C 180,E1 -11835.789,E2 -11835.789} C_VEL
LIN {X 0,Y 382.961,Z 331.408,A -85,B 0,C 180,E1 -11838.801,E2 -11838.801} C_VEL
LIN {X 0,Y 382.99,Z 331.401,A -85,B 0,C 180,E1 -11842.099,E2 -11842.099} C_VEL
LIN {X 0,Y 383.017,Z 331.396,A -85,B 0,C 180,E1 -11845.332,E2 -11845.332} C_VEL
LIN {X 0,Y 382.982,Z 331.402,A -85,B 0,C 180,E1 -11849.082,E2 -11849.082} C_VEL
LIN {X 0,Y 382.97,Z 331.406,A -85,B 0,C 180,E1 -11852.692,E2 -11852.692} C_VEL
LIN {X 0,Y 383.009,Z 331.401,A -85,B 0,C 180,E1 -11856.192,E2 -11856.192} C_VEL
LIN {X 0,Y 383.042,Z 331.393,A -85,B 0,C 180,E1 -11859.598,E2 -11859.598} C_VEL
LIN {X 0,Y 383.072,Z 331.39,A -85,B 0,C 180,E1 -11862.93,E2 -11862.93} C_VEL
LIN {X 0,Y 383.128,Z 331.386,A -85,B 0,C 180,E1 -11866.464,E2 -11866.464} C_VEL
LIN {X 0,Y 383.146,Z 331.383,A -85,B 0,C 180,E1 -11870.498,E2 -11870.498} C_VEL
LIN {X 0,Y 383.246,Z 331.37,A -85,B 0,C 180,E1 -11873.683,E2 -11873.683} C_VEL
LIN {X 0,Y 383.383,Z 331.356,A -85,B 0,C 180,E1 -11877.899,E2 -11877.899} C_VEL
LIN {X 0,Y 383.515,Z 331.341,A -85,B 0,C 180,E1 -11880,E2 -11880} C_VEL
LIN {X 0,Y 383.214,Z 331.372,A -85,B 0,C 180,E1 -11883.154,E2 -11883.154} C_VEL
LIN {X 0,Y 383.266,Z 331.367,A -85,B 0,C 180,E1 -11886.317,E2 -11886.317} C_VEL
LIN {X 0,Y 383.15,Z 331.382,A -85,B 0,C 180,E1 -11889.502,E2 -11889.502} C_VEL
LIN {X 0,Y 383.13,Z 331.386,A -85,B 0,C 180,E1 -11893.536,E2 -11893.536} C_VEL
LIN {X 0,Y 383.099,Z 331.39,A -85,B 0,C 180,E1 -11897.455,E2 -11897.455} C_VEL
LIN {X 0,Y 383.036,Z 331.394,A -85,B 0,C 180,E1 -11900.648,E2 -11900.648} C_VEL
LIN {X 0,Y 383.037,Z 331.398,A -85,B 0,C 180,E1 -11903.807,E2 -11903.807} C_VEL
LIN {X 0,Y 383.084,Z 331.389,A -85,B 0,C 180,E1 -11906.123,E2 -11906.123} C_VEL
LIN {X 0,Y 382.997,Z 331.403,A -85,B 0,C 180,E1 -11909.7,E2 -11909.7} C_VEL
LIN {X 0,Y 383.007,Z 331.404,A -85,B 0,C 180,E1 -11913.401,E2 -11913.401} C_VEL
LIN {X 0,Y 383.036,Z 331.394,A -85,B 0,C 180,E1 -11916.164,E2 -11916.164} C_VEL
LIN {X 0,Y 383.013,Z 331.397,A -85,B 0,C 180,E1 -11919.958,E2 -11919.958} C_VEL
LIN {X 0,Y 383.01,Z 331.399,A -85,B 0,C 180,E1 -11922.778,E2 -11922.778} C_VEL
LIN {X 0,Y 383.002,Z 331.399,A -85,B 0,C 180,E1 -11925.789,E2 -11925.789} C_VEL
LIN {X 0,Y 382.992,Z 331.402,A -85,B 0,C 180,E1 -11928.796,E2 -11928.796} C_VEL
LIN {X 0,Y 383.003,Z 331.398,A -85,B 0,C 180,E1 -11932.096,E2 -11932.096} C_VEL
LIN {X 0,Y 383.022,Z 331.399,A -85,B 0,C 180,E1 -11935.332,E2 -11935.332} C_VEL
LIN {X 0,Y 383.025,Z 331.417,A -85,B 0,C 180,E1 -11938.277,E2 -11938.277} C_VEL
LIN {X 0,Y 385.792,Z 343.767,A -85,B 0,C 180,E1 -11940.977,E2 -11940.977} C_VEL
LIN {X 0,Y 387.911,Z 353.642,A -85,B 0,C 180,E1 -11943.067,E2 -11943.067} C_VEL
LIN {X 0,Y 387.257,Z 362.753,A -85,B 0,C 180,E1 -11944.812,E2 -11944.812} C_VEL
LIN {X 0,Y 387.066,Z 365.211,A -85,B 0,C 180,E1 -11945.28,E2 -11945.28} C_VEL
LIN {X 0,Y 392.928,Z 400.818,A -85,B 0,C 180,E1 -11946.317,E2 -11946.317} C_VEL
LIN {X 0,Y 391.12,Z 503.867,A -85,B 0,C 180,E1 -11948.246,E2 -11948.246} C_VEL
LIN {X 0,Y 390.417,Z 518.415,A -85,B 0,C 180,E1 -11948.725,E2 -11948.725} C_VEL
LIN {X 0,Y 389.479,Z 532.383,A -85,B 0,C 180,E1 -11949.397,E2 -11949.397} C_VEL
LIN {X 0,Y 388.54,Z 545.028,A -85,B 0,C 180,E1 -11950.213,E2 -11950.213} C_VEL
LIN {X 0,Y 387.417,Z 557.332,A -85,B 0,C 180,E1 -11951.215,E2 -11951.215} C_VEL
LIN {X 0,Y 386.209,Z 568.991,A -85,B 0,C 180,E1 -11952.389,E2 -11952.389} C_VEL
LIN {X 0,Y 385.244,Z 578.7,A -85,B 0,C 180,E1 -11953.574,E2 -11953.574} C_VEL
LIN {X 0,Y 384.183,Z 589.476,A -85,B 0,C 180,E1 -11955.16,E2 -11955.16} C_VEL
LIN {X 0,Y 383.451,Z 598.37,A -85,B 0,C 180,E1 -11956.755,E2 -11956.755} C_VEL
LIN {X 0,Y 382.633,Z 606.874,A -85,B 0,C 180,E1 -11958.611,E2 -11958.611} C_VEL
LIN {X 0,Y 382.082,Z 613.704,A -85,B 0,C 180,E1 -11960.47,E2 -11960.47} C_VEL
LIN {X 0,Y 381.811,Z 618.389,A -85,B 0,C 180,E1 -11962.064,E2 -11962.064} C_VEL
LIN {X 0,Y 381.691,Z 622.605,A -85,B 0,C 180,E1 -11963.877,E2 -11963.877} C_VEL
LIN {X 0,Y 381.612,Z 625.828,A -85,B 0,C 180,E1 -11965.774,E2 -11965.774} C_VEL
LIN {X 0,Y 381.637,Z 628.074,A -85,B 0,C 180,E1 -11967.888,E2 -11967.888} C_VEL
LIN {X 0,Y 381.656,Z 628.95,A -85,B 0,C 180,E1 -11969.999,E2 -11969.999} C_VEL
LIN {X 0,Y 381.598,Z 628.478,A -85,B 0,C 180,E1 -11972.11,E2 -11972.11} C_VEL
LIN {X 0,Y 381.61,Z 626.665,A -85,B 0,C 180,E1 -11974.224,E2 -11974.224} C_VEL
LIN {X 0,Y 381.71,Z 623.477,A -85,B 0,C 180,E1 -11976.341,E2 -11976.341} C_VEL
LIN {X 0,Y 381.925,Z 618.806,A -85,B 0,C 180,E1 -11978.464,E2 -11978.464} C_VEL
LIN {X 0,Y 382.392,Z 612.498,A -85,B 0,C 180,E1 -11980.59,E2 -11980.59} C_VEL
LIN {X 0,Y 383.231,Z 605.503,A -85,B 0,C 180,E1 -11982.443,E2 -11982.443} C_VEL
LIN {X 0,Y 384.103,Z 597.066,A -85,B 0,C 180,E1 -11984.259,E2 -11984.259} C_VEL
LIN {X 0,Y 385.2,Z 587.877,A -85,B 0,C 180,E1 -11985.882,E2 -11985.882} C_VEL
LIN {X 0,Y 386.365,Z 578.975,A -85,B 0,C 180,E1 -11987.192,E2 -11987.192} C_VEL
LIN {X 0,Y 387.865,Z 567.223,A -85,B 0,C 180,E1 -11988.623,E2 -11988.623} C_VEL
LIN {X 0,Y 389.279,Z 555.471,A -85,B 0,C 180,E1 -11989.785,E2 -11989.785} C_VEL
LIN {X 0,Y 390.627,Z 542.258,A -85,B 0,C 180,E1 -11990.835,E2 -11990.835} C_VEL
LIN {X 0,Y 391.794,Z 529.087,A -85,B 0,C 180,E1 -11991.644,E2 -11991.644} C_VEL
LIN {X 0,Y 392.852,Z 515.016,A -85,B 0,C 180,E1 -11992.273,E2 -11992.273} C_VEL
LIN {X 0,Y 393.602,Z 501.551,A -85,B 0,C 180,E1 -11992.678,E2 -11992.678} C_VEL
LIN {X 0,Y 395.645,Z 401.31,A -85,B 0,C 180,E1 -11994.581,E2 -11994.581} C_VEL
LIN {X 0,Y 391.743,Z 378.887,A -85,B 0,C 180,E1 -11995.346,E2 -11995.346} C_VEL
LIN {X 0,Y 388.594,Z 364.473,A -85,B 0,C 180,E1 -11995.918,E2 -11995.918} C_VEL
LIN {X 0,Y 389.22,Z 358.327,A -85,B 0,C 180,E1 -11997.139,E2 -11997.139} C_VEL
LIN {X 0,Y 387.285,Z 348.268,A -85,B 0,C 180,E1 -11999.419,E2 -11999.419} C_VEL
LIN {X 0,Y 384.636,Z 337.6,A -85,B 0,C 180,E1 -12001.996,E2 -12001.996} C_VEL
LIN {X 0,Y 383.036,Z 331.394,A -85,B 0,C 180,E1 -12003.59,E2 -12003.59} C_VEL
LIN {X 0,Y 383.004,Z 331.404,A -85,B 0,C 180,E1 -12007.266,E2 -12007.266} C_VEL
LIN {X 0,Y 383.015,Z 331.401,A -85,B 0,C 180,E1 -12009.956,E2 -12009.956} C_VEL
LIN {X 0,Y 383.028,Z 331.393,A -85,B 0,C 180,E1 -12012.782,E2 -12012.782} C_VEL
LIN {X 0,Y 382.994,Z 331.39,A -85,B 0,C 180,E1 -12015.788,E2 -12015.788} C_VEL
LIN {X 0,Y 382.99,Z 331.399,A -85,B 0,C 180,E1 -12018.794,E2 -12018.794} C_VEL
LIN {X 0,Y 382.995,Z 331.398,A -85,B 0,C 180,E1 -12022.095,E2 -12022.095} C_VEL
LIN {X 0,Y 383.012,Z 331.399,A -85,B 0,C 180,E1 -12025.331,E2 -12025.331} C_VEL
LIN {X 0,Y 382.981,Z 331.402,A -85,B 0,C 180,E1 -12029.081,E2 -12029.081} C_VEL
LIN {X 0,Y 383.05,Z 331.392,A -85,B 0,C 180,E1 -12032.697,E2 -12032.697} C_VEL
LIN {X 0,Y 383.044,Z 331.395,A -85,B 0,C 180,E1 -12035.039,E2 -12035.039} C_VEL
LIN {X 0,Y 382.991,Z 331.405,A -85,B 0,C 180,E1 -12038.469,E2 -12038.469} C_VEL
LIN {X 0,Y 383.056,Z 331.39,A -85,B 0,C 180,E1 -12041.826,E2 -12041.826} C_VEL
LIN {X 0,Y 383.105,Z 331.379,A -85,B 0,C 180,E1 -12045.118,E2 -12045.118} C_VEL
LIN {X 0,Y 383.087,Z 331.383,A -85,B 0,C 180,E1 -12048.357,E2 -12048.357} C_VEL
LIN {X 0,Y 383.295,Z 331.363,A -85,B 0,C 180,E1 -12051.933,E2 -12051.933} C_VEL
LIN {X 0,Y 383.183,Z 331.377,A -85,B 0,C 180,E1 -12054.738,E2 -12054.738} C_VEL
LIN {X 0,Y 383.366,Z 331.352,A -85,B 0,C 180,E1 -12057.898,E2 -12057.898} C_VEL
LIN {X 0,Y 383.369,Z 331.354,A -85,B 0,C 180,E1 -12062.101,E2 -12062.101} C_VEL
LIN {X 0,Y 383.207,Z 331.374,A -85,B 0,C 180,E1 -12066.47,E2 -12066.47} C_VEL
LIN {X 0,Y 383.128,Z 331.382,A -85,B 0,C 180,E1 -12069.502,E2 -12069.502} C_VEL
LIN {X 0,Y 383.116,Z 331.386,A -85,B 0,C 180,E1 -12073.536,E2 -12073.536} C_VEL
LIN {X 0,Y 383.066,Z 331.396,A -85,B 0,C 180,E1 -12077.445,E2 -12077.445} C_VEL
LIN {X 0,Y 383.019,Z 331.398,A -85,B 0,C 180,E1 -12080.647,E2 -12080.647} C_VEL
LIN {X 0,Y 383.006,Z 331.401,A -85,B 0,C 180,E1 -12083.809,E2 -12083.809} C_VEL
LIN {X 0,Y 382.977,Z 331.4,A -85,B 0,C 180,E1 -12087.308,E2 -12087.308} C_VEL
LIN {X 0,Y 382.972,Z 331.411,A -85,B 0,C 180,E1 -12090.919,E2 -12090.919} C_VEL
LIN {X 0,Y 383.009,Z 331.405,A -85,B 0,C 180,E1 -12094.668,E2 -12094.668} C_VEL
LIN {X 0,Y 382.989,Z 331.405,A -85,B 0,C 180,E1 -12097.904,E2 -12097.904} C_VEL
LIN {X 0,Y 382.975,Z 331.403,A -85,B 0,C 180,E1 -12101.348,E2 -12101.348} C_VEL
LIN {X 0,Y 383.025,Z 331.497,A -85,B 0,C 180,E1 -12103.477,E2 -12103.477} C_VEL
LIN {X 0,Y 385.091,Z 339.967,A -85,B 0,C 180,E1 -12105.846,E2 -12105.846} C_VEL
LIN {X 0,Y 393.988,Z 359.543,A -85,B 0,C 180,E1 -12107,E2 -12107} C_VEL
LIN {X 0,Y 395.742,Z 364.485,A -85,B 0,C 180,E1 -12107.241,E2 -12107.241} C_VEL
LIN {X 0,Y 396.307,Z 367.137,A -85,B 0,C 180,E1 -12107.34,E2 -12107.34} C_VEL
LIN {X 0,Y 393.933,Z 476.174,A -85,B 0,C 180,E1 -12109.413,E2 -12109.413} C_VEL
LIN {X 0,Y 393.315,Z 490.262,A -85,B 0,C 180,E1 -12109.882,E2 -12109.882} C_VEL
LIN {X 0,Y 392.516,Z 502.653,A -85,B 0,C 180,E1 -12110.468,E2 -12110.468} C_VEL
LIN {X 0,Y 391.559,Z 515.096,A -85,B 0,C 180,E1 -12111.249,E2 -12111.249} C_VEL
LIN {X 0,Y 390.297,Z 527.68,A -85,B 0,C 180,E1 -12112.251,E2 -12112.251} C_VEL
LIN {X 0,Y 388.983,Z 539.282,A -85,B 0,C 180,E1 -12113.401,E2 -12113.401} C_VEL
LIN {X 0,Y 387.589,Z 550.695,A -85,B 0,C 180,E1 -12114.794,E2 -12114.794} C_VEL
LIN {X 0,Y 386.292,Z 560.781,A -85,B 0,C 180,E1 -12116.298,E2 -12116.298} C_VEL
LIN {X 0,Y 385.002,Z 570.353,A -85,B 0,C 180,E1 -12118.038,E2 -12118.038} C_VEL
LIN {X 0,Y 383.956,Z 578.298,A -85,B 0,C 180,E1 -12119.816,E2 -12119.816} C_VEL
LIN {X 0,Y 383.136,Z 585.073,A -85,B 0,C 180,E1 -12121.699,E2 -12121.699} C_VEL
LIN {X 0,Y 382.578,Z 589.559,A -85,B 0,C 180,E1 -12123.253,E2 -12123.253} C_VEL
LIN {X 0,Y 382.154,Z 593.55,A -85,B 0,C 180,E1 -12124.978,E2 -12124.978} C_VEL
LIN {X 0,Y 381.761,Z 597.319,A -85,B 0,C 180,E1 -12127.258,E2 -12127.258} C_VEL
LIN {X 0,Y 381.537,Z 599.495,A -85,B 0,C 180,E1 -12129.515,E2 -12129.515} C_VEL
LIN {X 0,Y 381.435,Z 600.156,A -85,B 0,C 180,E1 -12131.747,E2 -12131.747} C_VEL
LIN {X 0,Y 381.484,Z 599.342,A -85,B 0,C 180,E1 -12133.959,E2 -12133.959} C_VEL
LIN {X 0,Y 381.583,Z 597.113,A -85,B 0,C 180,E1 -12136.148,E2 -12136.148} C_VEL
LIN {X 0,Y 381.909,Z 593.428,A -85,B 0,C 180,E1 -12138.322,E2 -12138.322} C_VEL
LIN {X 0,Y 382.306,Z 588.22,A -85,B 0,C 180,E1 -12140.478,E2 -12140.478} C_VEL
LIN {X 0,Y 382.892,Z 582.158,A -85,B 0,C 180,E1 -12142.378,E2 -12142.378} C_VEL
LIN {X 0,Y 383.531,Z 574.804,A -85,B 0,C 180,E1 -12144.217,E2 -12144.217} C_VEL
LIN {X 0,Y 384.372,Z 567.009,A -85,B 0,C 180,E1 -12145.807,E2 -12145.807} C_VEL
LIN {X 0,Y 385.368,Z 557.641,A -85,B 0,C 180,E1 -12147.388,E2 -12147.388} C_VEL
LIN {X 0,Y 386.415,Z 547.288,A -85,B 0,C 180,E1 -12148.829,E2 -12148.829} C_VEL
LIN {X 0,Y 387.532,Z 535.873,A -85,B 0,C 180,E1 -12150.131,E2 -12150.131} C_VEL
LIN {X 0,Y 388.513,Z 524.826,A -85,B 0,C 180,E1 -12151.167,E2 -12151.167} C_VEL
LIN {X 0,Y 389.482,Z 512.949,A -85,B 0,C 180,E1 -12152.069,E2 -12152.069} C_VEL
LIN {X 0,Y 390.306,Z 500.029,A -85,B 0,C 180,E1 -12152.839,E2 -12152.839} C_VEL
LIN {X 0,Y 390.921,Z 486.96,A -85,B 0,C 180,E1 -12153.421,E2 -12153.421} C_VEL
LIN {X 0,Y 390.78,Z 481.247,A -85,B 0,C 180,E1 -12153.637,E2 -12153.637} C_VEL
LIN {X 0,Y 388.403,Z 471.98,A -85,B 0,C 180,E1 -12154.013,E2 -12154.013} C_VEL
LIN {X 0,Y 385.729,Z 462.659,A -85,B 0,C 180,E1 -12154.347,E2 -12154.347} C_VEL
LIN {X 0,Y 385.098,Z 456.847,A -85,B 0,C 180,E1 -12154.492,E2 -12154.492} C_VEL
LIN {X 0,Y 386.731,Z 366.876,A -85,B 0,C 180,E1 -12156.183,E2 -12156.183} C_VEL
LIN {X 0,Y 384.794,Z 358.981,A -85,B 0,C 180,E1 -12156.453,E2 -12156.453} C_VEL
LIN {X 0,Y 377.633,Z 339.383,A -85,B 0,C 180,E1 -12157.285,E2 -12157.285} C_VEL
LIN {X 0,Y 376.127,Z 332.26,A -85,B 0,C 180,E1 -12159.14,E2 -12159.14} C_VEL
LIN {X 0,Y 376.102,Z 332.261,A -85,B 0,C 180,E1 -12162.959,E2 -12162.959} C_VEL
LIN {X 0,Y 376.023,Z 332.267,A -85,B 0,C 180,E1 -12166.282,E2 -12166.282} C_VEL
LIN {X 0,Y 375.995,Z 332.272,A -85,B 0,C 180,E1 -12169.662,E2 -12169.662} C_VEL
LIN {X 0,Y 375.972,Z 332.275,A -85,B 0,C 180,E1 -12173.66,E2 -12173.66} C_VEL
LIN {X 0,Y 375.91,Z 332.284,A -85,B 0,C 180,E1 -12176.661,E2 -12176.661} C_VEL
LIN {X 0,Y 375.912,Z 332.287,A -85,B 0,C 180,E1 -12179.085,E2 -12179.085} C_VEL
LIN {X 0,Y 375.934,Z 332.279,A -85,B 0,C 180,E1 -12181.565,E2 -12181.565} C_VEL
LIN {X 0,Y 375.973,Z 332.277,A -85,B 0,C 180,E1 -12184.667,E2 -12184.667} C_VEL
LIN {X 0,Y 375.933,Z 332.28,A -85,B 0,C 180,E1 -12188.263,E2 -12188.263} C_VEL
LIN {X 0,Y 375.913,Z 332.281,A -85,B 0,C 180,E1 -12191.598,E2 -12191.598} C_VEL
LIN {X 0,Y 375.92,Z 332.287,A -85,B 0,C 180,E1 -12194.731,E2 -12194.731} C_VEL
LIN {X 0,Y 375.907,Z 332.282,A -85,B 0,C 180,E1 -12197.697,E2 -12197.697} C_VEL
LIN {X 0,Y 375.932,Z 332.284,A -85,B 0,C 180,E1 -12200.534,E2 -12200.534} C_VEL
LIN {X 0,Y 375.961,Z 332.275,A -85,B 0,C 180,E1 -12203.497,E2 -12203.497} C_VEL
LIN {X 0,Y 375.959,Z 332.276,A -85,B 0,C 180,E1 -12205.889,E2 -12205.889} C_VEL
LIN {X 0,Y 375.962,Z 332.275,A -85,B 0,C 180,E1 -12209.688,E2 -12209.688} C_VEL
LIN {X 0,Y 375.918,Z 332.283,A -85,B 0,C 180,E1 -12212.136,E2 -12212.136} C_VEL
LIN {X 0,Y 375.937,Z 332.283,A -85,B 0,C 180,E1 -12214.534,E2 -12214.534} C_VEL
LIN {X 0,Y 375.972,Z 332.275,A -85,B 0,C 180,E1 -12216.887,E2 -12216.887} C_VEL
LIN {X 0,Y 375.986,Z 332.278,A -85,B 0,C 180,E1 -12220.339,E2 -12220.339} C_VEL
LIN {X 0,Y 375.977,Z 332.274,A -85,B 0,C 180,E1 -12223.717,E2 -12223.717} C_VEL
LIN {X 0,Y 376.106,Z 332.257,A -85,B 0,C 180,E1 -12227.043,E2 -12227.043} C_VEL
LIN {X 0,Y 376.116,Z 332.26,A -85,B 0,C 180,E1 -12230.319,E2 -12230.319} C_VEL
LIN {X 0,Y 376.204,Z 332.246,A -85,B 0,C 180,E1 -12233.565,E2 -12233.565} C_VEL
LIN {X 0,Y 376.348,Z 332.231,A -85,B 0,C 180,E1 -12237.86,E2 -12237.86} C_VEL
LIN {X 0,Y 376.484,Z 332.217,A -85,B 0,C 180,E1 -12240,E2 -12240} C_VEL
LIN {X 0,Y 376.346,Z 332.232,A -85,B 0,C 180,E1 -12242.141,E2 -12242.141} C_VEL
LIN {X 0,Y 376.223,Z 332.244,A -85,B 0,C 180,E1 -12246.436,E2 -12246.436} C_VEL
LIN {X 0,Y 376.119,Z 332.26,A -85,B 0,C 180,E1 -12249.682,E2 -12249.682} C_VEL
LIN {X 0,Y 376.094,Z 332.264,A -85,B 0,C 180,E1 -12253.658,E2 -12253.658} C_VEL
LIN {X 0,Y 376.048,Z 332.27,A -85,B 0,C 180,E1 -12257.607,E2 -12257.607} C_VEL
LIN {X 0,Y 375.983,Z 332.272,A -85,B 0,C 180,E1 -12260.832,E2 -12260.832} C_VEL
LIN {X 0,Y 375.998,Z 332.271,A -85,B 0,C 180,E1 -12264.282,E2 -12264.282} C_VEL
LIN {X 0,Y 376.024,Z 332.267,A -85,B 0,C 180,E1 -12266.652,E2 -12266.652} C_VEL
LIN {X 0,Y 375.969,Z 332.274,A -85,B 0,C 180,E1 -12270.313,E2 -12270.313} C_VEL
LIN {X 0,Y 375.964,Z 332.275,A -85,B 0,C 180,E1 -12274.111,E2 -12274.111} C_VEL
LIN {X 0,Y 375.957,Z 332.276,A -85,B 0,C 180,E1 -12276.741,E2 -12276.741} C_VEL
LIN {X 0,Y 375.993,Z 332.272,A -85,B 0,C 180,E1 -12279.97,E2 -12279.97} C_VEL
LIN {X 0,Y 375.936,Z 332.28,A -85,B 0,C 180,E1 -12283.765,E2 -12283.765} C_VEL
LIN {X 0,Y 375.938,Z 332.28,A -85,B 0,C 180,E1 -12286.81,E2 -12286.81} C_VEL
LIN {X 0,Y 375.966,Z 332.275,A -85,B 0,C 180,E1 -12290.537,E2 -12290.537} C_VEL
LIN {X 0,Y 375.968,Z 332.277,A -85,B 0,C 180,E1 -12293.495,E2 -12293.495} C_VEL
LIN {X 0,Y 375.964,Z 332.275,A -85,B 0,C 180,E1 -12295.888,E2 -12295.888} C_VEL
LIN {X 0,Y 375.999,Z 332.431,A -85,B 0,C 180,E1 -12297.969,E2 -12297.969} C_VEL
LIN {X 0,Y 378.953,Z 345.561,A -85,B 0,C 180,E1 -12300.899,E2 -12300.899} C_VEL
LIN {X 0,Y 380.894,Z 354.492,A -85,B 0,C 180,E1 -12302.827,E2 -12302.827} C_VEL
LIN {X 0,Y 380.793,Z 358.938,A -85,B 0,C 180,E1 -12303.707,E2 -12303.707} C_VEL
LIN {X 0,Y 380.246,Z 364.941,A -85,B 0,C 180,E1 -12304.868,E2 -12304.868} C_VEL
LIN {X 0,Y 386.269,Z 401.71,A -85,B 0,C 180,E1 -12305.968,E2 -12305.968} C_VEL
LIN {X 0,Y 384.398,Z 503.865,A -85,B 0,C 180,E1 -12307.916,E2 -12307.916} C_VEL
LIN {X 0,Y 383.672,Z 518.336,A -85,B 0,C 180,E1 -12308.402,E2 -12308.402} C_VEL
LIN {X 0,Y 382.682,Z 532.261,A -85,B 0,C 180,E1 -12309.085,E2 -12309.085} C_VEL
LIN {X 0,Y 381.676,Z 545.526,A -85,B 0,C 180,E1 -12309.962,E2 -12309.962} C_VEL
LIN {X 0,Y 380.495,Z 557.901,A -85,B 0,C 180,E1 -12311.001,E2 -12311.001} C_VEL
LIN {X 0,Y 379.252,Z 569.423,A -85,B 0,C 180,E1 -12312.195,E2 -12312.195} C_VEL
LIN {X 0,Y 378.153,Z 580.012,A -85,B 0,C 180,E1 -12313.535,E2 -12313.535} C_VEL
LIN {X 0,Y 377.098,Z 590.535,A -85,B 0,C 180,E1 -12315.151,E2 -12315.151} C_VEL
LIN {X 0,Y 376.334,Z 599.349,A -85,B 0,C 180,E1 -12316.805,E2 -12316.805} C_VEL
LIN {X 0,Y 375.513,Z 607.462,A -85,B 0,C 180,E1 -12318.666,E2 -12318.666} C_VEL
LIN {X 0,Y 375.035,Z 613.264,A -85,B 0,C 180,E1 -12320.289,E2 -12320.289} C_VEL
LIN {X 0,Y 374.743,Z 617.982,A -85,B 0,C 180,E1 -12321.913,E2 -12321.913} C_VEL
LIN {X 0,Y 374.611,Z 622.498,A -85,B 0,C 180,E1 -12323.893,E2 -12323.893} C_VEL
LIN {X 0,Y 374.538,Z 625.491,A -85,B 0,C 180,E1 -12325.695,E2 -12325.695} C_VEL
LIN {X 0,Y 374.536,Z 627.766,A -85,B 0,C 180,E1 -12327.848,E2 -12327.848} C_VEL
LIN {X 0,Y 374.588,Z 628.674,A -85,B 0,C 180,E1 -12329.999,E2 -12329.999} C_VEL
LIN {X 0,Y 374.496,Z 628.23,A -85,B 0,C 180,E1 -12332.15,E2 -12332.15} C_VEL
LIN {X 0,Y 374.513,Z 626.446,A -85,B 0,C 180,E1 -12334.304,E2 -12334.304} C_VEL
LIN {X 0,Y 374.628,Z 623.287,A -85,B 0,C 180,E1 -12336.462,E2 -12336.462} C_VEL
LIN {X 0,Y 374.852,Z 618.663,A -85,B 0,C 180,E1 -12338.625,E2 -12338.625} C_VEL
LIN {X 0,Y 375.363,Z 612.403,A -85,B 0,C 180,E1 -12340.79,E2 -12340.79} C_VEL
LIN {X 0,Y 376.246,Z 605.46,A -85,B 0,C 180,E1 -12342.677,E2 -12342.677} C_VEL
LIN {X 0,Y 377.213,Z 596.882,A -85,B 0,C 180,E1 -12344.566,E2 -12344.566} C_VEL
LIN {X 0,Y 378.355,Z 587.949,A -85,B 0,C 180,E1 -12346.177,E2 -12346.177} C_VEL
LIN {X 0,Y 379.571,Z 579.116,A -85,B 0,C 180,E1 -12347.509,E2 -12347.509} C_VEL
LIN {X 0,Y 381.144,Z 567.446,A -85,B 0,C 180,E1 -12348.964,E2 -12348.964} C_VEL
LIN {X 0,Y 382.628,Z 555.8,A -85,B 0,C 180,E1 -12350.144,E2 -12350.144} C_VEL
LIN {X 0,Y 384.008,Z 542.894,A -85,B 0,C 180,E1 -12351.199,E2 -12351.199} C_VEL
LIN {X 0,Y 385.238,Z 529.787,A -85,B 0,C 180,E1 -12352.031,E2 -12352.031} C_VEL
LIN {X 0,Y 386.397,Z 515.417,A -85,B 0,C 180,E1 -12352.701,E2 -12352.701} C_VEL
LIN {X 0,Y 387.24,Z 500.955,A -85,B 0,C 180,E1 -12353.142,E2 -12353.142} C_VEL
LIN {X 0,Y 389.364,Z 402.404,A -85,B 0,C 180,E1 -12355.046,E2 -12355.046} C_VEL
LIN {X 0,Y 385.502,Z 380.237,A -85,B 0,C 180,E1 -12355.824,E2 -12355.824} C_VEL
LIN {X 0,Y 382.055,Z 364.115,A -85,B 0,C 180,E1 -12356.491,E2 -12356.491} C_VEL
LIN {X 0,Y 382.42,Z 359.907,A -85,B 0,C 180,E1 -12357.35,E2 -12357.35} C_VEL
LIN {X 0,Y 380.4,Z 349.652,A -85,B 0,C 180,E1 -12359.733,E2 -12359.733} C_VEL
LIN {X 0,Y 377.114,Z 336.544,A -85,B 0,C 180,E1 -12363.004,E2 -12363.004} C_VEL
LIN {X 0,Y 375.977,Z 332.274,A -85,B 0,C 180,E1 -12364.178,E2 -12364.178} C_VEL
LIN {X 0,Y 375.956,Z 332.276,A -85,B 0,C 180,E1 -12366.739,E2 -12366.739} C_VEL
LIN {X 0,Y 375.994,Z 332.275,A -85,B 0,C 180,E1 -12369.971,E2 -12369.971} C_VEL
LIN {X 0,Y 375.935,Z 332.283,A -85,B 0,C 180,E1 -12373.763,E2 -12373.763} C_VEL
LIN {X 0,Y 375.929,Z 332.275,A -85,B 0,C 180,E1 -12376.809,E2 -12376.809} C_VEL
LIN {X 0,Y 375.958,Z 332.264,A -85,B 0,C 180,E1 -12380.537,E2 -12380.537} C_VEL
LIN {X 0,Y 375.959,Z 332.277,A -85,B 0,C 180,E1 -12383.494,E2 -12383.494} C_VEL
LIN {X 0,Y 375.954,Z 332.28,A -85,B 0,C 180,E1 -12385.888,E2 -12385.888} C_VEL
LIN {X 0,Y 375.962,Z 332.276,A -85,B 0,C 180,E1 -12389.687,E2 -12389.687} C_VEL
LIN {X 0,Y 375.996,Z 332.276,A -85,B 0,C 180,E1 -12392.141,E2 -12392.141} C_VEL
LIN {X 0,Y 375.999,Z 332.273,A -85,B 0,C 180,E1 -12394.538,E2 -12394.538} C_VEL
LIN {X 0,Y 375.955,Z 332.275,A -85,B 0,C 180,E1 -12398.045,E2 -12398.045} C_VEL
LIN {X 0,Y 376.002,Z 332.265,A -85,B 0,C 180,E1 -12401.473,E2 -12401.473} C_VEL
LIN {X 0,Y 376.053,Z 332.258,A -85,B 0,C 180,E1 -12404.832,E2 -12404.832} C_VEL
LIN {X 0,Y 376.04,Z 332.263,A -85,B 0,C 180,E1 -12408.136,E2 -12408.136} C_VEL
LIN {X 0,Y 376.249,Z 332.241,A -85,B 0,C 180,E1 -12411.878,E2 -12411.878} C_VEL
LIN {X 0,Y 376.156,Z 332.253,A -85,B 0,C 180,E1 -12414.639,E2 -12414.639} C_VEL
LIN {X 0,Y 376.331,Z 332.228,A -85,B 0,C 180,E1 -12417.859,E2 -12417.859} C_VEL
LIN {X 0,Y 376.334,Z 332.231,A -85,B 0,C 180,E1 -12422.14,E2 -12422.14} C_VEL
LIN {X 0,Y 376.178,Z 332.249,A -85,B 0,C 180,E1 -12426.455,E2 -12426.455} C_VEL
LIN {X 0,Y 376.099,Z 332.258,A -85,B 0,C 180,E1 -12429.682,E2 -12429.682} C_VEL
LIN {X 0,Y 376.08,Z 332.263,A -85,B 0,C 180,E1 -12433.657,E2 -12433.657} C_VEL
LIN {X 0,Y 376.017,Z 332.274,A -85,B 0,C 180,E1 -12437.599,E2 -12437.599} C_VEL
LIN {X 0,Y 375.969,Z 332.278,A -85,B 0,C 180,E1 -12440.832,E2 -12440.832} C_VEL
LIN {X 0,Y 375.963,Z 332.277,A -85,B 0,C 180,E1 -12444.283,E2 -12444.283} C_VEL
LIN {X 0,Y 375.919,Z 332.275,A -85,B 0,C 180,E1 -12447.864,E2 -12447.864} C_VEL
LIN {X 0,Y 375.948,Z 332.282,A -85,B 0,C 180,E1 -12451.562,E2 -12451.562} C_VEL
LIN {X 0,Y 375.948,Z 332.283,A -85,B 0,C 180,E1 -12455.416,E2 -12455.416} C_VEL
LIN {X 0,Y 375.963,Z 332.281,A -85,B 0,C 180,E1 -12458.271,E2 -12458.271} C_VEL
LIN {X 0,Y 375.925,Z 332.279,A -85,B 0,C 180,E1 -12461.601,E2 -12461.601} C_VEL
LIN {X 0,Y 375.988,Z 332.377,A -85,B 0,C 180,E1 -12462.946,E2 -12462.946} C_VEL
LIN {X 0,Y 377.945,Z 340.273,A -85,B 0,C 180,E1 -12465.214,E2 -12465.214} C_VEL
LIN {X 0,Y 386.841,Z 359.419,A -85,B 0,C 180,E1 -12466.414,E2 -12466.414} C_VEL
LIN {X 0,Y 389.695,Z 366.708,A -85,B 0,C 180,E1 -12466.803,E2 -12466.803} C_VEL
LIN {X 0,Y 390.049,Z 369.181,A -85,B 0,C 180,E1 -12466.883,E2 -12466.883} C_VEL
LIN {X 0,Y 387.59,Z 476.244,A -85,B 0,C 180,E1 -12468.95,E2 -12468.95} C_VEL
LIN {X 0,Y 386.895,Z 490.878,A -85,B 0,C 180,E1 -12469.446,E2 -12469.446} C_VEL
LIN {X 0,Y 385.957,Z 504.655,A -85,B 0,C 180,E1 -12470.129,E2 -12470.129} C_VEL
LIN {X 0,Y 384.902,Z 517.175,A -85,B 0,C 180,E1 -12470.956,E2 -12470.956} C_VEL
LIN {X 0,Y 383.569,Z 529.54,A -85,B 0,C 180,E1 -12471.986,E2 -12471.986} C_VEL
LIN {X 0,Y 382.061,Z 542.008,A -85,B 0,C 180,E1 -12473.286,E2 -12473.286} C_VEL
LIN {X 0,Y 380.762,Z 552.135,A -85,B 0,C 180,E1 -12474.584,E2 -12474.584} C_VEL
LIN {X 0,Y 379.296,Z 562.743,A -85,B 0,C 180,E1 -12476.231,E2 -12476.231} C_VEL
LIN {X 0,Y 377.992,Z 571.996,A -85,B 0,C 180,E1 -12478.003,E2 -12478.003} C_VEL
LIN {X 0,Y 376.926,Z 579.528,A -85,B 0,C 180,E1 -12479.774,E2 -12479.774} C_VEL
LIN {X 0,Y 376.039,Z 586.335,A -85,B 0,C 180,E1 -12481.775,E2 -12481.775} C_VEL
LIN {X 0,Y 375.498,Z 590.554,A -85,B 0,C 180,E1 -12483.309,E2 -12483.309} C_VEL
LIN {X 0,Y 375.061,Z 594.356,A -85,B 0,C 180,E1 -12485.065,E2 -12485.065} C_VEL
LIN {X 0,Y 374.741,Z 597.187,A -85,B 0,C 180,E1 -12486.808,E2 -12486.808} C_VEL
LIN {X 0,Y 374.478,Z 599.546,A -85,B 0,C 180,E1 -12489.111,E2 -12489.111} C_VEL
LIN {X 0,Y 374.339,Z 600.408,A -85,B 0,C 180,E1 -12491.389,E2 -12491.389} C_VEL
LIN {X 0,Y 374.397,Z 599.818,A -85,B 0,C 180,E1 -12493.647,E2 -12493.647} C_VEL
LIN {X 0,Y 374.463,Z 597.78,A -85,B 0,C 180,E1 -12495.879,E2 -12495.879} C_VEL
LIN {X 0,Y 374.776,Z 594.274,A -85,B 0,C 180,E1 -12498.097,E2 -12498.097} C_VEL
LIN {X 0,Y 375.065,Z 590.692,A -85,B 0,C 180,E1 -12499.747,E2 -12499.747} C_VEL
LIN {X 0,Y 375.483,Z 586.126,A -85,B 0,C 180,E1 -12501.389,E2 -12501.389} C_VEL
LIN {X 0,Y 376.079,Z 579.562,A -85,B 0,C 180,E1 -12503.294,E2 -12503.294} C_VEL
LIN {X 0,Y 376.946,Z 571.414,A -85,B 0,C 180,E1 -12505.188,E2 -12505.188} C_VEL
LIN {X 0,Y 377.839,Z 562.897,A -85,B 0,C 180,E1 -12506.802,E2 -12506.802} C_VEL
LIN {X 0,Y 378.961,Z 552.583,A -85,B 0,C 180,E1 -12508.407,E2 -12508.407} C_VEL
LIN {X 0,Y 380.172,Z 541.327,A -85,B 0,C 180,E1 -12509.836,E2 -12509.836} C_VEL
LIN {X 0,Y 381.265,Z 529.568,A -85,B 0,C 180,E1 -12511.057,E2 -12511.057} C_VEL
LIN {X 0,Y 382.391,Z 516.953,A -85,B 0,C 180,E1 -12512.107,E2 -12512.107} C_VEL
LIN {X 0,Y 383.388,Z 503.927,A -85,B 0,C 180,E1 -12512.956,E2 -12512.956} C_VEL
LIN {X 0,Y 384.068,Z 490.05,A -85,B 0,C 180,E1 -12513.64,E2 -12513.64} C_VEL
LIN {X 0,Y 384.677,Z 475.359,A -85,B 0,C 180,E1 -12514.126,E2 -12514.126} C_VEL
LIN {X 0,Y 385.098,Z 456.847,A -85,B 0,C 180,E1 -12514.492,E2 -12514.492} C_VEL
LIN {X 0,Y 384.544,Z 451.043,A -85,B 0,C 180,E1 -12514.636,E2 -12514.636} C_VEL
LIN {X 0,Y 379.592,Z 432.329,A -85,B 0,C 180,E1 -12515.28,E2 -12515.28} C_VEL
LIN {X 0,Y 379.028,Z 426.526,A -85,B 0,C 180,E1 -12515.429,E2 -12515.429} C_VEL
LIN {X 0,Y 380.13,Z 368.552,A -85,B 0,C 180,E1 -12516.536,E2 -12516.536} C_VEL
LIN {X 0,Y 378.627,Z 361.787,A -85,B 0,C 180,E1 -12516.762,E2 -12516.762} C_VEL
LIN {X 0,Y 370.462,Z 339.548,A -85,B 0,C 180,E1 -12517.758,E2 -12517.758} C_VEL
LIN {X 0,Y 369.075,Z 333.139,A -85,B 0,C 180,E1 -12519.454,E2 -12519.454} C_VEL
LIN {X 0,Y 369.036,Z 333.139,A -85,B 0,C 180,E1 -12523.773,E2 -12523.773} C_VEL
LIN {X 0,Y 368.99,Z 333.145,A -85,B 0,C 180,E1 -12527.744,E2 -12527.744} C_VEL
LIN {X 0,Y 368.908,Z 333.159,A -85,B 0,C 180,E1 -12531.222,E2 -12531.222} C_VEL
LIN {X 0,Y 368.921,Z 333.155,A -85,B 0,C 180,E1 -12534.779,E2 -12534.779} C_VEL
LIN {X 0,Y 368.891,Z 333.16,A -85,B 0,C 180,E1 -12538.793,E2 -12538.793} C_VEL
LIN {X 0,Y 368.888,Z 333.157,A -85,B 0,C 180,E1 -12542.24,E2 -12542.24} C_VEL
LIN {X 0,Y 368.922,Z 333.157,A -85,B 0,C 180,E1 -12545.001,E2 -12545.001} C_VEL
LIN {X 0,Y 368.875,Z 333.162,A -85,B 0,C 180,E1 -12548.634,E2 -12548.634} C_VEL
LIN {X 0,Y 368.858,Z 333.16,A -85,B 0,C 180,E1 -12552.006,E2 -12552.006} C_VEL
LIN {X 0,Y 368.873,Z 333.16,A -85,B 0,C 180,E1 -12555.175,E2 -12555.175} C_VEL
LIN {X 0,Y 368.86,Z 333.161,A -85,B 0,C 180,E1 -12558.175,E2 -12558.175} C_VEL
LIN {X 0,Y 368.874,Z 333.158,A -85,B 0,C 180,E1 -12561.367,E2 -12561.367} C_VEL
LIN {X 0,Y 368.935,Z 333.151,A -85,B 0,C 180,E1 -12565.147,E2 -12565.147} C_VEL
LIN {X 0,Y 368.914,Z 333.154,A -85,B 0,C 180,E1 -12569.046,E2 -12569.046} C_VEL
LIN {X 0,Y 368.908,Z 333.154,A -85,B 0,C 180,E1 -12571.558,E2 -12571.558} C_VEL
LIN {X 0,Y 368.921,Z 333.154,A -85,B 0,C 180,E1 -12574.014,E2 -12574.014} C_VEL
LIN {X 0,Y 368.898,Z 333.155,A -85,B 0,C 180,E1 -12577.603,E2 -12577.603} C_VEL
LIN {X 0,Y 368.932,Z 333.151,A -85,B 0,C 180,E1 -12581.105,E2 -12581.105} C_VEL
LIN {X 0,Y 368.942,Z 333.153,A -85,B 0,C 180,E1 -12584.533,E2 -12584.533} C_VEL
LIN {X 0,Y 369.061,Z 333.136,A -85,B 0,C 180,E1 -12586.791,E2 -12586.791} C_VEL
LIN {X 0,Y 369.066,Z 333.14,A -85,B 0,C 180,E1 -12590.132,E2 -12590.132} C_VEL
LIN {X 0,Y 369.164,Z 333.122,A -85,B 0,C 180,E1 -12593.441,E2 -12593.441} C_VEL
LIN {X 0,Y 369.312,Z 333.107,A -85,B 0,C 180,E1 -12597.819,E2 -12597.819} C_VEL
LIN {X 0,Y 369.433,Z 333.095,A -85,B 0,C 180,E1 -12600,E2 -12600} C_VEL
LIN {X 0,Y 369.31,Z 333.107,A -85,B 0,C 180,E1 -12602.182,E2 -12602.182} C_VEL
LIN {X 0,Y 369.182,Z 333.12,A -85,B 0,C 180,E1 -12606.559,E2 -12606.559} C_VEL
LIN {X 0,Y 369.069,Z 333.14,A -85,B 0,C 180,E1 -12609.869,E2 -12609.869} C_VEL
LIN {X 0,Y 369.041,Z 333.144,A -85,B 0,C 180,E1 -12613.772,E2 -12613.772} C_VEL
LIN {X 0,Y 369.006,Z 333.147,A -85,B 0,C 180,E1 -12617.768,E2 -12617.768} C_VEL
LIN {X 0,Y 368.935,Z 333.153,A -85,B 0,C 180,E1 -12621.22,E2 -12621.22} C_VEL
LIN {X 0,Y 368.962,Z 333.147,A -85,B 0,C 180,E1 -12624.775,E2 -12624.775} C_VEL
LIN {X 0,Y 368.967,Z 333.149,A -85,B 0,C 180,E1 -12627.203,E2 -12627.203} C_VEL
LIN {X 0,Y 368.934,Z 333.152,A -85,B 0,C 180,E1 -12630.953,E2 -12630.953} C_VEL
LIN {X 0,Y 368.933,Z 333.153,A -85,B 0,C 180,E1 -12635.001,E2 -12635.001} C_VEL
LIN {X 0,Y 368.913,Z 333.154,A -85,B 0,C 180,E1 -12638.64,E2 -12638.64} C_VEL
LIN {X 0,Y 368.886,Z 333.157,A -85,B 0,C 180,E1 -12642.009,E2 -12642.009} C_VEL
LIN {X 0,Y 368.931,Z 333.157,A -85,B 0,C 180,E1 -12645.183,E2 -12645.183} C_VEL
LIN {X 0,Y 368.886,Z 333.156,A -85,B 0,C 180,E1 -12648.177,E2 -12648.177} C_VEL
LIN {X 0,Y 368.913,Z 333.157,A -85,B 0,C 180,E1 -12651.359,E2 -12651.359} C_VEL
LIN {X 0,Y 368.941,Z 333.155,A -85,B 0,C 180,E1 -12655.146,E2 -12655.146} C_VEL
LIN {X 0,Y 368.957,Z 333.342,A -85,B 0,C 180,E1 -12657.631,E2 -12657.631} C_VEL
LIN {X 0,Y 371.867,Z 346.215,A -85,B 0,C 180,E1 -12660.568,E2 -12660.568} C_VEL
LIN {X 0,Y 374.085,Z 356.953,A -85,B 0,C 180,E1 -12662.926,E2 -12662.926} C_VEL
LIN {X 0,Y 373.448,Z 364.997,A -85,B 0,C 180,E1 -12664.476,E2 -12664.476} C_VEL
LIN {X 0,Y 379.609,Z 402.913,A -85,B 0,C 180,E1 -12665.613,E2 -12665.613} C_VEL
LIN {X 0,Y 377.68,Z 502.635,A -85,B 0,C 180,E1 -12667.538,E2 -12667.538} C_VEL
LIN {X 0,Y 377.036,Z 516.693,A -85,B 0,C 180,E1 -12668.003,E2 -12668.003} C_VEL
LIN {X 0,Y 376.022,Z 530.974,A -85,B 0,C 180,E1 -12668.696,E2 -12668.696} C_VEL
LIN {X 0,Y 374.942,Z 544.489,A -85,B 0,C 180,E1 -12669.589,E2 -12669.589} C_VEL
LIN {X 0,Y 373.674,Z 556.979,A -85,B 0,C 180,E1 -12670.64,E2 -12670.64} C_VEL
LIN {X 0,Y 372.465,Z 568.626,A -85,B 0,C 180,E1 -12671.859,E2 -12671.859} C_VEL
LIN {X 0,Y 371.285,Z 579.302,A -85,B 0,C 180,E1 -12673.221,E2 -12673.221} C_VEL
LIN {X 0,Y 370.151,Z 589.9,A -85,B 0,C 180,E1 -12674.866,E2 -12674.866} C_VEL
LIN {X 0,Y 369.355,Z 598.904,A -85,B 0,C 180,E1 -12676.574,E2 -12676.574} C_VEL
LIN {X 0,Y 368.502,Z 606.98,A -85,B 0,C 180,E1 -12678.447,E2 -12678.447} C_VEL
LIN {X 0,Y 367.979,Z 612.807,A -85,B 0,C 180,E1 -12680.101,E2 -12680.101} C_VEL
LIN {X 0,Y 367.664,Z 617.568,A -85,B 0,C 180,E1 -12681.756,E2 -12681.756} C_VEL
LIN {X 0,Y 367.505,Z 622.465,A -85,B 0,C 180,E1 -12683.949,E2 -12683.949} C_VEL
LIN {X 0,Y 367.444,Z 625.151,A -85,B 0,C 180,E1 -12685.611,E2 -12685.611} C_VEL
LIN {X 0,Y 367.435,Z 627.458,A -85,B 0,C 180,E1 -12687.807,E2 -12687.807} C_VEL
LIN {X 0,Y 367.505,Z 628.397,A -85,B 0,C 180,E1 -12689.999,E2 -12689.999} C_VEL
LIN {X 0,Y 367.396,Z 627.983,A -85,B 0,C 180,E1 -12692.192,E2 -12692.192} C_VEL
LIN {X 0,Y 367.421,Z 626.231,A -85,B 0,C 180,E1 -12694.387,E2 -12694.387} C_VEL
LIN {X 0,Y 367.556,Z 623.109,A -85,B 0,C 180,E1 -12696.587,E2 -12696.587} C_VEL
LIN {X 0,Y 367.795,Z 618.531,A -85,B 0,C 180,E1 -12698.792,E2 -12698.792} C_VEL
LIN {X 0,Y 368.185,Z 614.018,A -85,B 0,C 180,E1 -12700.447,E2 -12700.447} C_VEL
LIN {X 0,Y 369.005,Z 607.542,A -85,B 0,C 180,E1 -12702.371,E2 -12702.371} C_VEL
LIN {X 0,Y 369.933,Z 599.402,A -85,B 0,C 180,E1 -12704.326,E2 -12704.326} C_VEL
LIN {X 0,Y 371.07,Z 591.172,A -85,B 0,C 180,E1 -12705.939,E2 -12705.939} C_VEL
LIN {X 0,Y 372.504,Z 581.148,A -85,B 0,C 180,E1 -12707.569,E2 -12707.569} C_VEL
LIN {X 0,Y 374.158,Z 570.026,A -85,B 0,C 180,E1 -12709.047,E2 -12709.047} C_VEL
LIN {X 0,Y 375.825,Z 557.6,A -85,B 0,C 180,E1 -12710.382,E2 -12710.382} C_VEL
LIN {X 0,Y 377.249,Z 545.476,A -85,B 0,C 180,E1 -12711.432,E2 -12711.432} C_VEL
LIN {X 0,Y 378.484,Z 532.836,A -85,B 0,C 180,E1 -12712.301,E2 -12712.301} C_VEL
LIN {X 0,Y 379.77,Z 518.158,A -85,B 0,C 180,E1 -12713.048,E2 -12713.048} C_VEL
LIN {X 0,Y 380.722,Z 504.306,A -85,B 0,C 180,E1 -12713.526,E2 -12713.526} C_VEL
LIN {X 0,Y 381.453,Z 476.765,A -85,B 0,C 180,E1 -12714.103,E2 -12714.103} C_VEL
LIN {X 0,Y 383.067,Z 403.014,A -85,B 0,C 180,E1 -12715.54,E2 -12715.54} C_VEL
LIN {X 0,Y 378.922,Z 379.228,A -85,B 0,C 180,E1 -12716.406,E2 -12716.406} C_VEL
LIN {X 0,Y 375.468,Z 363.929,A -85,B 0,C 180,E1 -12717.055,E2 -12717.055} C_VEL
LIN {X 0,Y 375.603,Z 361.416,A -85,B 0,C 180,E1 -12717.586,E2 -12717.586} C_VEL
LIN {X 0,Y 373.503,Z 351.072,A -85,B 0,C 180,E1 -12720.053,E2 -12720.053} C_VEL
LIN {X 0,Y 370.279,Z 338.115,A -85,B 0,C 180,E1 -12723.37,E2 -12723.37} C_VEL
LIN {X 0,Y 368.935,Z 333.156,A -85,B 0,C 180,E1 -12724.769,E2 -12724.769} C_VEL
LIN {X 0,Y 368.912,Z 333.15,A -85,B 0,C 180,E1 -12728.641,E2 -12728.641} C_VEL
LIN {X 0,Y 368.906,Z 333.148,A -85,B 0,C 180,E1 -12731.817,E2 -12731.817} C_VEL
LIN {X 0,Y 368.877,Z 333.151,A -85,B 0,C 180,E1 -12735.175,E2 -12735.175} C_VEL
LIN {X 0,Y 368.882,Z 333.162,A -85,B 0,C 180,E1 -12738.177,E2 -12738.177} C_VEL
LIN {X 0,Y 368.904,Z 333.148,A -85,B 0,C 180,E1 -12741.358,E2 -12741.358} C_VEL
LIN {X 0,Y 368.931,Z 333.154,A -85,B 0,C 180,E1 -12745.146,E2 -12745.146} C_VEL
LIN {X 0,Y 368.923,Z 333.153,A -85,B 0,C 180,E1 -12749.046,E2 -12749.046} C_VEL
LIN {X 0,Y 368.98,Z 333.146,A -85,B 0,C 180,E1 -12751.564,E2 -12751.564} C_VEL
LIN {X 0,Y 368.993,Z 333.141,A -85,B 0,C 180,E1 -12754.019,E2 -12754.019} C_VEL
LIN {X 0,Y 368.92,Z 333.147,A -85,B 0,C 180,E1 -12757.604,E2 -12757.604} C_VEL
LIN {X 0,Y 368.951,Z 333.143,A -85,B 0,C 180,E1 -12761.105,E2 -12761.105} C_VEL
LIN {X 0,Y 368.993,Z 333.138,A -85,B 0,C 180,E1 -12764.535,E2 -12764.535} C_VEL
LIN {X 0,Y 368.996,Z 333.143,A -85,B 0,C 180,E1 -12767.906,E2 -12767.906} C_VEL
LIN {X 0,Y 369.22,Z 333.117,A -85,B 0,C 180,E1 -12771.801,E2 -12771.801} C_VEL
LIN {X 0,Y 369.13,Z 333.128,A -85,B 0,C 180,E1 -12774.537,E2 -12774.537} C_VEL
LIN {X 0,Y 369.295,Z 333.104,A -85,B 0,C 180,E1 -12777.818,E2 -12777.818} C_VEL
LIN {X 0,Y 369.298,Z 333.107,A -85,B 0,C 180,E1 -12782.181,E2 -12782.181} C_VEL
LIN {X 0,Y 369.142,Z 333.126,A -85,B 0,C 180,E1 -12786.559,E2 -12786.559} C_VEL
LIN {X 0,Y 369.05,Z 333.138,A -85,B 0,C 180,E1 -12789.868,E2 -12789.868} C_VEL
LIN {X 0,Y 369.028,Z 333.143,A -85,B 0,C 180,E1 -12793.772,E2 -12793.772} C_VEL
LIN {X 0,Y 368.968,Z 333.15,A -85,B 0,C 180,E1 -12797.757,E2 -12797.757} C_VEL
LIN {X 0,Y 368.9,Z 333.159,A -85,B 0,C 180,E1 -12801.221,E2 -12801.221} C_VEL
LIN {X 0,Y 368.917,Z 333.155,A -85,B 0,C 180,E1 -12804.778,E2 -12804.778} C_VEL
LIN {X 0,Y 368.887,Z 333.147,A -85,B 0,C 180,E1 -12808.793,E2 -12808.793} C_VEL
LIN {X 0,Y 368.889,Z 333.157,A -85,B 0,C 180,E1 -12812.238,E2 -12812.238} C_VEL
LIN {X 0,Y 368.92,Z 333.163,A -85,B 0,C 180,E1 -12815.002,E2 -12815.002} C_VEL
LIN {X 0,Y 368.898,Z 333.158,A -85,B 0,C 180,E1 -12818.64,E2 -12818.64} C_VEL
LIN {X 0,Y 368.906,Z 333.154,A -85,B 0,C 180,E1 -12822.335,E2 -12822.335} C_VEL
LIN {X 0,Y 370.777,Z 340.662,A -85,B 0,C 180,E1 -12824.562,E2 -12824.562} C_VEL
LIN {X 0,Y 379.154,Z 358.054,A -85,B 0,C 180,E1 -12825.721,E2 -12825.721} C_VEL
LIN {X 0,Y 383.673,Z 368.81,A -85,B 0,C 180,E1 -12826.348,E2 -12826.348} C_VEL
LIN {X 0,Y 383.653,Z 377.422,A -85,B 0,C 180,E1 -12826.531,E2 -12826.531} C_VEL
LIN {X 0,Y 381.265,Z 476.189,A -85,B 0,C 180,E1 -12828.465,E2 -12828.465} C_VEL
LIN {X 0,Y 380.583,Z 490.607,A -85,B 0,C 180,E1 -12828.954,E2 -12828.954} C_VEL
LIN {X 0,Y 379.624,Z 503.987,A -85,B 0,C 180,E1 -12829.614,E2 -12829.614} C_VEL
LIN {X 0,Y 378.451,Z 517.391,A -85,B 0,C 180,E1 -12830.505,E2 -12830.505} C_VEL
LIN {X 0,Y 377.103,Z 529.36,A -85,B 0,C 180,E1 -12831.512,E2 -12831.512} C_VEL
LIN {X 0,Y 375.654,Z 540.946,A -85,B 0,C 180,E1 -12832.723,E2 -12832.723} C_VEL
LIN {X 0,Y 374.088,Z 552.373,A -85,B 0,C 180,E1 -12834.191,E2 -12834.191} C_VEL
LIN {X 0,Y 372.499,Z 563.304,A -85,B 0,C 180,E1 -12835.923,E2 -12835.923} C_VEL
LIN {X 0,Y 371.179,Z 572.209,A -85,B 0,C 180,E1 -12837.665,E2 -12837.665} C_VEL
LIN {X 0,Y 370.05,Z 579.754,A -85,B 0,C 180,E1 -12839.468,E2 -12839.468} C_VEL
LIN {X 0,Y 369.22,Z 585.402,A -85,B 0,C 180,E1 -12841.115,E2 -12841.115} C_VEL
LIN {X 0,Y 368.605,Z 590.033,A -85,B 0,C 180,E1 -12842.769,E2 -12842.769} C_VEL
LIN {X 0,Y 368.114,Z 594.04,A -85,B 0,C 180,E1 -12844.561,E2 -12844.561} C_VEL
LIN {X 0,Y 367.698,Z 597.341,A -85,B 0,C 180,E1 -12846.555,E2 -12846.555} C_VEL
LIN {X 0,Y 367.404,Z 599.604,A -85,B 0,C 180,E1 -12848.689,E2 -12848.689} C_VEL
LIN {X 0,Y 367.371,Z 600.304,A -85,B 0,C 180,E1 -12849.859,E2 -12849.859} C_VEL
LIN {X 0,Y 367.242,Z 600.611,A -85,B 0,C 180,E1 -12852.171,E2 -12852.171} C_VEL
LIN {X 0,Y 367.303,Z 600.222,A -85,B 0,C 180,E1 -12853.322,E2 -12853.322} C_VEL
LIN {X 0,Y 367.341,Z 598.39,A -85,B 0,C 180,E1 -12855.6,E2 -12855.6} C_VEL
LIN {X 0,Y 367.659,Z 595.104,A -85,B 0,C 180,E1 -12857.863,E2 -12857.863} C_VEL
LIN {X 0,Y 367.935,Z 591.619,A -85,B 0,C 180,E1 -12859.546,E2 -12859.546} C_VEL
LIN {X 0,Y 368.346,Z 587.238,A -85,B 0,C 180,E1 -12861.221,E2 -12861.221} C_VEL
LIN {X 0,Y 368.903,Z 581.832,A -85,B 0,C 180,E1 -12862.902,E2 -12862.902} C_VEL
LIN {X 0,Y 369.659,Z 574.202,A -85,B 0,C 180,E1 -12864.82,E2 -12864.82} C_VEL
LIN {X 0,Y 370.546,Z 566.192,A -85,B 0,C 180,E1 -12866.467,E2 -12866.467} C_VEL
LIN {X 0,Y 371.679,Z 556.525,A -85,B 0,C 180,E1 -12868.105,E2 -12868.105} C_VEL
LIN {X 0,Y 372.778,Z 546.319,A -85,B 0,C 180,E1 -12869.535,E2 -12869.535} C_VEL
LIN {X 0,Y 374.086,Z 533.988,A -85,B 0,C 180,E1 -12870.943,E2 -12870.943} C_VEL
LIN {X 0,Y 375.143,Z 522.399,A -85,B 0,C 180,E1 -12872.014,E2 -12872.014} C_VEL
LIN {X 0,Y 376.295,Z 508.767,A -85,B 0,C 180,E1 -12873.012,E2 -12873.012} C_VEL
LIN {X 0,Y 377.108,Z 495.693,A -85,B 0,C 180,E1 -12873.741,E2 -12873.741} C_VEL
LIN {X 0,Y 377.774,Z 481.542,A -85,B 0,C 180,E1 -12874.302,E2 -12874.302} C_VEL
LIN {X 0,Y 378.236,Z 465.051,A -85,B 0,C 180,E1 -12874.697,E2 -12874.697} C_VEL
LIN {X 0,Y 379.028,Z 426.526,A -85,B 0,C 180,E1 -12875.429,E2 -12875.429} C_VEL
LIN {X 0,Y 378.435,Z 420.722,A -85,B 0,C 180,E1 -12875.58,E2 -12875.58} C_VEL
LIN {X 0,Y 373.393,Z 402.045,A -85,B 0,C 180,E1 -12876.25,E2 -12876.25} C_VEL
LIN {X 0,Y 372.953,Z 396.239,A -85,B 0,C 180,E1 -12876.396,E2 -12876.396} C_VEL
LIN {X 0,Y 373.463,Z 369.057,A -85,B 0,C 180,E1 -12876.926,E2 -12876.926} C_VEL
LIN {X 0,Y 371.964,Z 363.17,A -85,B 0,C 180,E1 -12877.139,E2 -12877.139} C_VEL
LIN {X 0,Y 363.318,Z 339.892,A -85,B 0,C 180,E1 -12878.201,E2 -12878.201} C_VEL
LIN {X 0,Y 362.031,Z 334.017,A -85,B 0,C 180,E1 -12879.781,E2 -12879.781} C_VEL
LIN {X 0,Y 361.997,Z 334.015,A -85,B 0,C 180,E1 -12883.9,E2 -12883.9} C_VEL
LIN {X 0,Y 361.926,Z 334.027,A -85,B 0,C 180,E1 -12886.935,E2 -12886.935} C_VEL
LIN {X 0,Y 361.885,Z 334.029,A -85,B 0,C 180,E1 -12890.462,E2 -12890.462} C_VEL
LIN {X 0,Y 361.893,Z 334.027,A -85,B 0,C 180,E1 -12894.114,E2 -12894.114} C_VEL
LIN {X 0,Y 361.834,Z 334.035,A -85,B 0,C 180,E1 -12897.786,E2 -12897.786} C_VEL
LIN {X 0,Y 361.825,Z 334.039,A -85,B 0,C 180,E1 -12901.28,E2 -12901.28} C_VEL
LIN {X 0,Y 361.849,Z 334.034,A -85,B 0,C 180,E1 -12904.282,E2 -12904.282} C_VEL
LIN {X 0,Y 361.856,Z 334.035,A -85,B 0,C 180,E1 -12907.222,E2 -12907.222} C_VEL
LIN {X 0,Y 361.81,Z 334.044,A -85,B 0,C 180,E1 -12910.751,E2 -12910.751} C_VEL
LIN {X 0,Y 361.811,Z 334.04,A -85,B 0,C 180,E1 -12914.37,E2 -12914.37} C_VEL
LIN {X 0,Y 361.822,Z 334.036,A -85,B 0,C 180,E1 -12917.571,E2 -12917.571} C_VEL
LIN {X 0,Y 361.841,Z 334.034,A -85,B 0,C 180,E1 -12921.572,E2 -12921.572} C_VEL
LIN {X 0,Y 361.874,Z 334.036,A -85,B 0,C 180,E1 -12924.656,E2 -12924.656} C_VEL
LIN {X 0,Y 361.839,Z 334.039,A -85,B 0,C 180,E1 -12928.371,E2 -12928.371} C_VEL
LIN {X 0,Y 361.868,Z 334.032,A -85,B 0,C 180,E1 -12930.953,E2 -12930.953} C_VEL
LIN {X 0,Y 361.853,Z 334.036,A -85,B 0,C 180,E1 -12934.705,E2 -12934.705} C_VEL
LIN {X 0,Y 361.855,Z 334.039,A -85,B 0,C 180,E1 -12938.345,E2 -12938.345} C_VEL
LIN {X 0,Y 361.92,Z 334.028,A -85,B 0,C 180,E1 -12942.087,E2 -12942.087} C_VEL
LIN {X 0,Y 361.982,Z 334.022,A -85,B 0,C 180,E1 -12946.114,E2 -12946.114} C_VEL
LIN {X 0,Y 362.003,Z 334.018,A -85,B 0,C 180,E1 -12949.938,E2 -12949.938} C_VEL
LIN {X 0,Y 362.127,Z 333.999,A -85,B 0,C 180,E1 -12953.313,E2 -12953.313} C_VEL
LIN {X 0,Y 362.275,Z 333.984,A -85,B 0,C 180,E1 -12957.777,E2 -12957.777} C_VEL
LIN {X 0,Y 362.384,Z 333.973,A -85,B 0,C 180,E1 -12960,E2 -12960} C_VEL
LIN {X 0,Y 362.274,Z 333.984,A -85,B 0,C 180,E1 -12962.224,E2 -12962.224} C_VEL
LIN {X 0,Y 362.143,Z 333.997,A -85,B 0,C 180,E1 -12966.687,E2 -12966.687} C_VEL
LIN {X 0,Y 362.005,Z 334.017,A -85,B 0,C 180,E1 -12970.063,E2 -12970.063} C_VEL
LIN {X 0,Y 362.002,Z 334.019,A -85,B 0,C 180,E1 -12973.899,E2 -12973.899} C_VEL
LIN {X 0,Y 361.972,Z 334.021,A -85,B 0,C 180,E1 -12977.939,E2 -12977.939} C_VEL
LIN {X 0,Y 361.898,Z 334.033,A -85,B 0,C 180,E1 -12981.653,E2 -12981.653} C_VEL
LIN {X 0,Y 361.933,Z 334.026,A -85,B 0,C 180,E1 -12985.29,E2 -12985.29} C_VEL
LIN {X 0,Y 361.913,Z 334.029,A -85,B 0,C 180,E1 -12987.779,E2 -12987.779} C_VEL
LIN {X 0,Y 361.842,Z 334.038,A -85,B 0,C 180,E1 -12991.629,E2 -12991.629} C_VEL
LIN {X 0,Y 361.878,Z 334.035,A -85,B 0,C 180,E1 -12995.345,E2 -12995.345} C_VEL
LIN {X 0,Y 361.874,Z 334.033,A -85,B 0,C 180,E1 -12999.026,E2 -12999.026} C_VEL
LIN {X 0,Y 361.841,Z 334.036,A -85,B 0,C 180,E1 -13002.828,E2 -13002.828} C_VEL
LIN {X 0,Y 361.839,Z 334.035,A -85,B 0,C 180,E1 -13005.944,E2 -13005.944} C_VEL
LIN {X 0,Y 361.84,Z 334.04,A -85,B 0,C 180,E1 -13009.244,E2 -13009.244} C_VEL
LIN {X 0,Y 361.868,Z 334.034,A -85,B 0,C 180,E1 -13012.777,E2 -13012.777} C_VEL
LIN {X 0,Y 361.858,Z 334.033,A -85,B 0,C 180,E1 -13015.719,E2 -13015.719} C_VEL
LIN {X 0,Y 361.908,Z 334.198,A -85,B 0,C 180,E1 -13017.268,E2 -13017.268} C_VEL
LIN {X 0,Y 364.905,Z 347.356,A -85,B 0,C 180,E1 -13020.336,E2 -13020.336} C_VEL
LIN {X 0,Y 367.068,Z 357.634,A -85,B 0,C 180,E1 -13022.644,E2 -13022.644} C_VEL
LIN {X 0,Y 366.643,Z 364.243,A -85,B 0,C 180,E1 -13023.989,E2 -13023.989} C_VEL
LIN {X 0,Y 367.106,Z 367.368,A -85,B 0,C 180,E1 -13024.13,E2 -13024.13} C_VEL
LIN {X 0,Y 372.932,Z 402.922,A -85,B 0,C 180,E1 -13025.225,E2 -13025.225} C_VEL
LIN {X 0,Y 371.131,Z 498.178,A -85,B 0,C 180,E1 -13027.083,E2 -13027.083} C_VEL
LIN {X 0,Y 370.543,Z 513.081,A -85,B 0,C 180,E1 -13027.523,E2 -13027.523} C_VEL
LIN {X 0,Y 369.524,Z 527.207,A -85,B 0,C 180,E1 -13028.156,E2 -13028.156} C_VEL
LIN {X 0,Y 368.476,Z 540.49,A -85,B 0,C 180,E1 -13028.982,E2 -13028.982} C_VEL
LIN {X 0,Y 367.288,Z 553.163,A -85,B 0,C 180,E1 -13029.998,E2 -13029.998} C_VEL
LIN {X 0,Y 365.95,Z 565.45,A -85,B 0,C 180,E1 -13031.235,E2 -13031.235} C_VEL
LIN {X 0,Y 364.699,Z 576.618,A -85,B 0,C 180,E1 -13032.62,E2 -13032.62} C_VEL
LIN {X 0,Y 363.59,Z 585.959,A -85,B 0,C 180,E1 -13034.011,E2 -13034.011} C_VEL
LIN {X 0,Y 362.507,Z 595.753,A -85,B 0,C 180,E1 -13035.781,E2 -13035.781} C_VEL
LIN {X 0,Y 361.781,Z 603.09,A -85,B 0,C 180,E1 -13037.376,E2 -13037.376} C_VEL
LIN {X 0,Y 361.05,Z 610.495,A -85,B 0,C 180,E1 -13039.342,E2 -13039.342} C_VEL
LIN {X 0,Y 360.695,Z 615.677,A -85,B 0,C 180,E1 -13041.031,E2 -13041.031} C_VEL
LIN {X 0,Y 360.478,Z 621.025,A -85,B 0,C 180,E1 -13043.281,E2 -13043.281} C_VEL
LIN {X 0,Y 360.353,Z 624.801,A -85,B 0,C 180,E1 -13045.525,E2 -13045.525} C_VEL
LIN {X 0,Y 360.336,Z 627.145,A -85,B 0,C 180,E1 -13047.763,E2 -13047.763} C_VEL
LIN {X 0,Y 360.423,Z 628.119,A -85,B 0,C 180,E1 -13049.999,E2 -13049.999} C_VEL
LIN {X 0,Y 360.297,Z 627.738,A -85,B 0,C 180,E1 -13052.235,E2 -13052.235} C_VEL
LIN {X 0,Y 360.333,Z 626.021,A -85,B 0,C 180,E1 -13054.474,E2 -13054.474} C_VEL
LIN {X 0,Y 360.486,Z 622.933,A -85,B 0,C 180,E1 -13056.717,E2 -13056.717} C_VEL
LIN {X 0,Y 360.752,Z 618.394,A -85,B 0,C 180,E1 -13058.965,E2 -13058.965} C_VEL
LIN {X 0,Y 361.162,Z 613.918,A -85,B 0,C 180,E1 -13060.652,E2 -13060.652} C_VEL
LIN {X 0,Y 362.176,Z 606.473,A -85,B 0,C 180,E1 -13062.893,E2 -13062.893} C_VEL
LIN {X 0,Y 363.205,Z 598.283,A -85,B 0,C 180,E1 -13064.855,E2 -13064.855} C_VEL
LIN {X 0,Y 364.44,Z 589.753,A -85,B 0,C 180,E1 -13066.524,E2 -13066.524} C_VEL
LIN {X 0,Y 366.053,Z 579.461,A -85,B 0,C 180,E1 -13068.178,E2 -13068.178} C_VEL
LIN {X 0,Y 367.765,Z 567.99,A -85,B 0,C 180,E1 -13069.682,E2 -13069.682} C_VEL
LIN {X 0,Y 369.553,Z 555.179,A -85,B 0,C 180,E1 -13071.035,E2 -13071.035} C_VEL
LIN {X 0,Y 371.043,Z 542.502,A -85,B 0,C 180,E1 -13072.105,E2 -13072.105} C_VEL
LIN {X 0,Y 372.452,Z 529.165,A -85,B 0,C 180,E1 -13072.976,E2 -13072.976} C_VEL
LIN {X 0,Y 373.716,Z 514.759,A -85,B 0,C 180,E1 -13073.663,E2 -13073.663} C_VEL
LIN {X 0,Y 374.561,Z 500.257,A -85,B 0,C 180,E1 -13074.121,E2 -13074.121} C_VEL
LIN {X 0,Y 376.863,Z 404.029,A -85,B 0,C 180,E1 -13076.04,E2 -13076.04} C_VEL
LIN {X 0,Y 372.834,Z 380.945,A -85,B 0,C 180,E1 -13076.908,E2 -13076.908} C_VEL
LIN {X 0,Y 368.862,Z 363.537,A -85,B 0,C 180,E1 -13077.691,E2 -13077.691} C_VEL
LIN {X 0,Y 366.873,Z 353.577,A -85,B 0,C 180,E1 -13080.118,E2 -13080.118} C_VEL
LIN {X 0,Y 363.934,Z 341.556,A -85,B 0,C 180,E1 -13083.245,E2 -13083.245} C_VEL
LIN {X 0,Y 361.873,Z 334.032,A -85,B 0,C 180,E1 -13085.344,E2 -13085.344} C_VEL
LIN {X 0,Y 361.873,Z 334.027,A -85,B 0,C 180,E1 -13089.027,E2 -13089.027} C_VEL
LIN {X 0,Y 361.852,Z 334.027,A -85,B 0,C 180,E1 -13092.434,E2 -13092.434} C_VEL
LIN {X 0,Y 361.814,Z 334.027,A -85,B 0,C 180,E1 -13095.945,E2 -13095.945} C_VEL
LIN {X 0,Y 361.834,Z 334.031,A -85,B 0,C 180,E1 -13099.243,E2 -13099.243} C_VEL
LIN {X 0,Y 361.865,Z 334.036,A -85,B 0,C 180,E1 -13102.774,E2 -13102.774} C_VEL
LIN {X 0,Y 361.849,Z 334.036,A -85,B 0,C 180,E1 -13105.719,E2 -13105.719} C_VEL
LIN {X 0,Y 361.87,Z 334.032,A -85,B 0,C 180,E1 -13109.671,E2 -13109.671} C_VEL
LIN {X 0,Y 361.948,Z 334.018,A -85,B 0,C 180,E1 -13113.474,E2 -13113.474} C_VEL
LIN {X 0,Y 361.877,Z 334.024,A -85,B 0,C 180,E1 -13117.143,E2 -13117.143} C_VEL
LIN {X 0,Y 361.9,Z 334.022,A -85,B 0,C 180,E1 -13120.723,E2 -13120.723} C_VEL
LIN {X 0,Y 361.927,Z 334.025,A -85,B 0,C 180,E1 -13123.065,E2 -13123.065} C_VEL
LIN {X 0,Y 361.991,Z 334.019,A -85,B 0,C 180,E1 -13126.527,E2 -13126.527} C_VEL
LIN {X 0,Y 362.022,Z 334.01,A -85,B 0,C 180,E1 -13129.937,E2 -13129.937} C_VEL
LIN {X 0,Y 362.142,Z 333.994,A -85,B 0,C 180,E1 -13132.192,E2 -13132.192} C_VEL
LIN {X 0,Y 362.104,Z 334.004,A -85,B 0,C 180,E1 -13134.431,E2 -13134.431} C_VEL
LIN {X 0,Y 362.258,Z 333.98,A -85,B 0,C 180,E1 -13137.776,E2 -13137.776} C_VEL
LIN {X 0,Y 362.261,Z 333.984,A -85,B 0,C 180,E1 -13142.223,E2 -13142.223} C_VEL
LIN {X 0,Y 362.106,Z 334.002,A -85,B 0,C 180,E1 -13146.687,E2 -13146.687} C_VEL
LIN {X 0,Y 361.987,Z 334.019,A -85,B 0,C 180,E1 -13150.063,E2 -13150.063} C_VEL
LIN {X 0,Y 361.989,Z 334.02,A -85,B 0,C 180,E1 -13153.899,E2 -13153.899} C_VEL
LIN {X 0,Y 361.911,Z 334.028,A -85,B 0,C 180,E1 -13157.915,E2 -13157.915} C_VEL
LIN {X 0,Y 361.852,Z 334.032,A -85,B 0,C 180,E1 -13161.655,E2 -13161.655} C_VEL
LIN {X 0,Y 361.874,Z 334.033,A -85,B 0,C 180,E1 -13165.294,E2 -13165.294} C_VEL
LIN {X 0,Y 361.846,Z 334.025,A -85,B 0,C 180,E1 -13169.074,E2 -13169.074} C_VEL
LIN {X 0,Y 361.839,Z 334.03,A -85,B 0,C 180,E1 -13172.945,E2 -13172.945} C_VEL
LIN {X 0,Y 361.859,Z 334.037,A -85,B 0,C 180,E1 -13175.637,E2 -13175.637} C_VEL
LIN {X 0,Y 361.859,Z 334.031,A -85,B 0,C 180,E1 -13179.027,E2 -13179.027} C_VEL
LIN {X 0,Y 361.874,Z 334.227,A -85,B 0,C 180,E1 -13181.812,E2 -13181.812} C_VEL
LIN {X 0,Y 363.595,Z 340.888,A -85,B 0,C 180,E1 -13183.854,E2 -13183.854} C_VEL
LIN {X 0,Y 373.242,Z 360.674,A -85,B 0,C 180,E1 -13185.245,E2 -13185.245} C_VEL
